// TIA Portal project "DALU-Projekt_HMI_V19" (V19)

(* hardware
DEVICE "SIMATIC 1200-Station_3"  S71200.Device
   slot 0: "S7-1200 Baugruppenträger"  Rack  V1.0
   slot 1: "Target_3"  CPU 1214C DC/DC/DC  6ES7 214-1AE30-0XB0  V2.2
   slot 101: "Target 3 CM 1243-2"  CM 1243-2  3RK7243-2AA30-0XB0  V1.0
   slot 102: "Target 3 CM 1243-5"  CM 1243-5  6GK7 243-5DX30-0XE0  V1.0
DEVICE "ASi-3-S9 (4DI)"  AS-i slave
   slot 0: "-"  Rail
   slot 1: "ASi-3-S9 (4DI)"  AS-i Standard Slave  AS-i Standard Slave Universal
      slot 1: "ASi-3-S9 (4DI) [AS-i Slave (D)]"  AS-i Address-Module
      slot 2: "ASi-3-S9 (4DI) [AS-i Slave (A)]"  AS-i Address-Module
      slot 3: "ASi-3-S9 (4DI) [AS-i Slave (T)]"  AS-i Address-Module
DEVICE "ASi-3-S5 (2AI)"  AS-i slave
   slot 0: "-"  Rail
   slot 1: "ASi-3-S5 (2AI)"  AS-i K60, 2AI-C  3RK1 207-1BQ40-0AA3
      slot 1: "ASi-3-S5 (2AI) [AS-i Slave (D)]"  AS-i Address-Module
      slot 2: "ASi-3-S5 (2AI) [AS-i Slave (A)]"  AS-i Address-Module
      slot 3: "ASi-3-S5 (2AI) [AS-i Slave (T)]"  AS-i Address-Module
DEVICE "ASi-3-S1 (4DI/4DO)"  AS-i slave
   slot 0: "-"  Rail
   slot 1: "ASi-3-S1 (4DI/4DO)"  AS-i 3SB3, 4DI/4DO  3SF5 500-0BC
      slot 1: "ASi-3-S1 (4DI/4DO) [AS-i Slave (D)]"  AS-i Address-Module
      slot 2: "ASi-3-S1 (4DI/4DO) [AS-i Slave (A)]"  AS-i Address-Module
      slot 3: "ASi-3-S1 (4DI/4DO) [AS-i Slave (T)]"  AS-i Address-Module
DEVICE "ASi-3-S7 (2DI,2PO)"  AS-i slave
   slot 0: "-"  Rail
   slot 1: "ASi-3-S7 (2DI,2PO)"  AS-i Standard Slave  AS-i Standard Slave Universal
      slot 1: "ASi-3-S7 (2DI,2PO) [AS-i Slave (D)]"  AS-i Address-Module
      slot 2: "ASi-3-S7 (2DI,2PO) [AS-i Slave (A)]"  AS-i Address-Module
      slot 3: "ASi-3-S7 (2DI,2PO) [AS-i Slave (T)]"  AS-i Address-Module
DEVICE "ASi-3-S3 (2AI)"  AS-i slave
   slot 0: "-"  Rail
   slot 1: "ASi-3-S3 (2AI)"  AS-i K60, 2AI-V  3RK1 207-2BQ40-0AA3
      slot 1: "ASi-3-S3 (2AI) [AS-i Slave (D)]"  AS-i Address-Module
      slot 2: "ASi-3-S3 (2AI) [AS-i Slave (A)]"  AS-i Address-Module
      slot 3: "ASi-3-S3 (2AI) [AS-i Slave (T)]"  AS-i Address-Module
DEVICE "ASi-3-S8 (3DI/1DO)"  AS-i slave
   slot 0: "-"  Rail
   slot 1: "ASi-3-S8 (3DI/1DO)"  AS-i Standard Slave  AS-i Standard Slave Universal
      slot 1: "ASi-3-S8 (3DI/1DO) [AS-i Slave (D)]"  AS-i Address-Module
      slot 2: "ASi-3-S8 (3DI/1DO) [AS-i Slave (A)]"  AS-i Address-Module
      slot 3: "ASi-3-S8 (3DI/1DO) [AS-i Slave (T)]"  AS-i Address-Module
DEVICE "DP_3_S1"  GSD.Device
   slot 0: "Baugruppenträger"  Rail
   slot 0: "DP_3_Simodrive"  6FX2001-5xPxx  4.2
DEVICE "ASi-3-S2 (2AO)"  AS-i slave
   slot 0: "-"  Rail
   slot 1: "ASi-3-S2 (2AO)"  AS-i K60, 2AO-V  3RK1 107-2BQ40-0AA3
      slot 1: "ASi-3-S2 (2AO) [AS-i Slave (D)]"  AS-i Address-Module
      slot 2: "ASi-3-S2 (2AO) [AS-i Slave (A)]"  AS-i Address-Module
      slot 3: "ASi-3-S2 (2AO) [AS-i Slave (T)]"  AS-i Address-Module
DEVICE "ASi-3-S4 (4DI/4DO)"  AS-i slave
   slot 0: "-"  Rail
   slot 1: "ASi-3-S4 (4DI/4DO)"  AS-i K60, 4DI/4DO  3RK1 400-1DQ01-0AA3
      slot 1: "ASi-3-S4 (4DI/4DO) [AS-i Slave (D)]"  AS-i Address-Module
      slot 2: "ASi-3-S4 (4DI/4DO) [AS-i Slave (A)]"  AS-i Address-Module
      slot 3: "ASi-3-S4 (4DI/4DO) [AS-i Slave (T)]"  AS-i Address-Module
DEVICE "ASi-3-S6 (4DI)"  AS-i slave
   slot 0: "-"  Rail
   slot 1: "ASi-3-S6 (4DI)"  AS-i K45, 4DI  3RK1 200-0CQ20-0AA3
      slot 1: "ASi-3-S6 (4DI) [AS-i Slave (D)]"  AS-i Address-Module
      slot 2: "ASi-3-S6 (4DI) [AS-i Slave (A)]"  AS-i Address-Module
      slot 3: "ASi-3-S6 (4DI) [AS-i Slave (T)]"  AS-i Address-Module
DEVICE "SIMATIC 1200-Station_4"  S71200.Device
   slot 0: "S7-1200 Baugruppenträger"  Rack  V1.0
   slot 1: "Target_4"  CPU 1214C DC/DC/DC  6ES7 214-1AE30-0XB0  V2.2
   slot 101: "Target 4 CM 1243-2"  CM 1243-2  3RK7243-2AA30-0XB0  V1.0
   slot 102: "Target 4 CM 1243-5"  CM 1243-5  6GK7 243-5DX30-0XE0  V1.0
DEVICE "ASi-4-S9 (4DI)"  AS-i slave
   slot 0: "-"  Rail
   slot 1: "ASi-4-S9 (4DI)"  AS-i Standard Slave  AS-i Standard Slave Universal
      slot 1: "ASi-4-S9 (4DI) [AS-i Slave (D)]"  AS-i Address-Module
      slot 2: "ASi-4-S9 (4DI) [AS-i Slave (A)]"  AS-i Address-Module
      slot 3: "ASi-4-S9 (4DI) [AS-i Slave (T)]"  AS-i Address-Module
DEVICE "ASi-4-S5 (2AI)"  AS-i slave
   slot 0: "-"  Rail
   slot 1: "ASi-4-S5 (2AI)"  AS-i K60, 2AI-C  3RK1 207-1BQ40-0AA3
      slot 1: "ASi-4-S5 (2AI) [AS-i Slave (D)]"  AS-i Address-Module
      slot 2: "ASi-4-S5 (2AI) [AS-i Slave (A)]"  AS-i Address-Module
      slot 3: "ASi-4-S5 (2AI) [AS-i Slave (T)]"  AS-i Address-Module
DEVICE "ASi-4-S1 (4DI/4DO)"  AS-i slave
   slot 0: "-"  Rail
   slot 1: "ASi-4-S1 (4DI/4DO)"  AS-i 3SB3, 4DI/4DO  3SF5 500-0BC
      slot 1: "ASi-4-S1 (4DI/4DO) [AS-i Slave (D)]"  AS-i Address-Module
      slot 2: "ASi-4-S1 (4DI/4DO) [AS-i Slave (A)]"  AS-i Address-Module
      slot 3: "ASi-4-S1 (4DI/4DO) [AS-i Slave (T)]"  AS-i Address-Module
DEVICE "ASi-4-S7 (2DI,2PO)"  AS-i slave
   slot 0: "-"  Rail
   slot 1: "ASi-4-S7 (2DI,2PO)"  AS-i Standard Slave  AS-i Standard Slave Universal
      slot 1: "ASi-4-S7 (2DI,2PO) [AS-i Slave (D)]"  AS-i Address-Module
      slot 2: "ASi-4-S7 (2DI,2PO) [AS-i Slave (A)]"  AS-i Address-Module
      slot 3: "ASi-4-S7 (2DI,2PO) [AS-i Slave (T)]"  AS-i Address-Module
DEVICE "ASi-4-S3 (2AI)"  AS-i slave
   slot 0: "-"  Rail
   slot 1: "ASi-4-S3 (2AI)"  AS-i K60, 2AI-V  3RK1 207-2BQ40-0AA3
      slot 1: "ASi-4-S3 (2AI) [AS-i Slave (D)]"  AS-i Address-Module
      slot 2: "ASi-4-S3 (2AI) [AS-i Slave (A)]"  AS-i Address-Module
      slot 3: "ASi-4-S3 (2AI) [AS-i Slave (T)]"  AS-i Address-Module
DEVICE "ASi-4-S8 (3DI/1DO)"  AS-i slave
   slot 0: "-"  Rail
   slot 1: "ASi-4-S8 (3DI/1DO)"  AS-i Standard Slave  AS-i Standard Slave Universal
      slot 1: "ASi-4-S8 (3DI/1DO) [AS-i Slave (D)]"  AS-i Address-Module
      slot 2: "ASi-4-S8 (3DI/1DO) [AS-i Slave (A)]"  AS-i Address-Module
      slot 3: "ASi-4-S8 (3DI/1DO) [AS-i Slave (T)]"  AS-i Address-Module
DEVICE "DP_4_S1"  GSD.Device
   slot 0: "Baugruppenträger"  Rail
   slot 0: "DP_4_Simodrive"  6FX2001-5xPxx  4.2
DEVICE "ASi-4-S2 (2AO)"  AS-i slave
   slot 0: "-"  Rail
   slot 1: "ASi-4-S2 (2AO)"  AS-i K60, 2AO-V  3RK1 107-2BQ40-0AA3
      slot 1: "ASi-4-S2 (2AO) [AS-i Slave (D)]"  AS-i Address-Module
      slot 2: "ASi-4-S2 (2AO) [AS-i Slave (A)]"  AS-i Address-Module
      slot 3: "ASi-4-S2 (2AO) [AS-i Slave (T)]"  AS-i Address-Module
DEVICE "ASi-4-S4 (4DI/4DO)"  AS-i slave
   slot 0: "-"  Rail
   slot 1: "ASi-4-S4 (4DI/4DO)"  AS-i K60, 4DI/4DO  3RK1 400-1DQ01-0AA3
      slot 1: "ASi-4-S4 (4DI/4DO) [AS-i Slave (D)]"  AS-i Address-Module
      slot 2: "ASi-4-S4 (4DI/4DO) [AS-i Slave (A)]"  AS-i Address-Module
      slot 3: "ASi-4-S4 (4DI/4DO) [AS-i Slave (T)]"  AS-i Address-Module
DEVICE "ASi-4-S6 (4DI)"  AS-i slave
   slot 0: "-"  Rail
   slot 1: "ASi-4-S6 (4DI)"  AS-i K45, 4DI  3RK1 200-0CQ20-0AA3
      slot 1: "ASi-4-S6 (4DI) [AS-i Slave (D)]"  AS-i Address-Module
      slot 2: "ASi-4-S6 (4DI) [AS-i Slave (A)]"  AS-i Address-Module
      slot 3: "ASi-4-S6 (4DI) [AS-i Slave (T)]"  AS-i Address-Module
DEVICE "SIMATIC 1200-Station_5"  S71200.Device
   slot 0: "S7-1200 Baugruppenträger"  Rack  V1.0
   slot 1: "Target_5"  CPU 1214C DC/DC/DC  6ES7 214-1AE30-0XB0  V2.2
   slot 101: "Target 5 CM 1243-2"  CM 1243-2  3RK7243-2AA30-0XB0  V1.0
   slot 102: "Target 5 CM 1243-5"  CM 1243-5  6GK7 243-5DX30-0XE0  V1.0
   slot 103: "CM CANopen_1"  021620-B  V1.0
DEVICE "ASi-5-S9 (4DI)"  AS-i slave
   slot 0: "-"  Rail
   slot 1: "ASi-5-S9 (4DI)"  AS-i Standard Slave  AS-i Standard Slave Universal
      slot 1: "ASi-5-S9 (4DI) [AS-i Slave (D)]"  AS-i Address-Module
      slot 2: "ASi-5-S9 (4DI) [AS-i Slave (A)]"  AS-i Address-Module
      slot 3: "ASi-5-S9 (4DI) [AS-i Slave (T)]"  AS-i Address-Module
DEVICE "ASi-5-S5 (2AI)"  AS-i slave
   slot 0: "-"  Rail
   slot 1: "ASi-5-S5 (2AI)"  AS-i K60, 2AI-C  3RK1 207-1BQ40-0AA3
      slot 1: "ASi-5-S5 (2AI) [AS-i Slave (D)]"  AS-i Address-Module
      slot 2: "ASi-5-S5 (2AI) [AS-i Slave (A)]"  AS-i Address-Module
      slot 3: "ASi-5-S5 (2AI) [AS-i Slave (T)]"  AS-i Address-Module
DEVICE "ASi-5-S3 (2AI)"  AS-i slave
   slot 0: "-"  Rail
   slot 1: "ASi-5-S3 (2AI)"  AS-i K60, 2AI-V  3RK1 207-2BQ40-0AA3
      slot 1: "ASi-5-S3 (2AI) [AS-i Slave (D)]"  AS-i Address-Module
      slot 2: "ASi-5-S3 (2AI) [AS-i Slave (A)]"  AS-i Address-Module
      slot 3: "ASi-5-S3 (2AI) [AS-i Slave (T)]"  AS-i Address-Module
DEVICE "ASi-5-S7 (2DI,2PO)"  AS-i slave
   slot 0: "-"  Rail
   slot 1: "ASi-5-S7 (2DI,2PO)"  AS-i Standard Slave  AS-i Standard Slave Universal
      slot 1: "ASi-5-S7 (2DI,2PO) [AS-i Slave (D)]"  AS-i Address-Module
      slot 2: "ASi-5-S7 (2DI,2PO) [AS-i Slave (A)]"  AS-i Address-Module
      slot 3: "ASi-5-S7 (2DI,2PO) [AS-i Slave (T)]"  AS-i Address-Module
DEVICE "ASi-5-S2 (2AO)"  AS-i slave
   slot 0: "-"  Rail
   slot 1: "ASi-5-S2 (2AO)"  AS-i K60, 2AO-V  3RK1 107-2BQ40-0AA3
      slot 1: "ASi-5-S2 (2AO) [AS-i Slave (D)]"  AS-i Address-Module
      slot 2: "ASi-5-S2 (2AO) [AS-i Slave (A)]"  AS-i Address-Module
      slot 3: "ASi-5-S2 (2AO) [AS-i Slave (T)]"  AS-i Address-Module
DEVICE "ASi-5-S8 (3DI/1DO)"  AS-i slave
   slot 0: "-"  Rail
   slot 1: "ASi-5-S8 (3DI/1DO)"  AS-i Standard Slave  AS-i Standard Slave Universal
      slot 1: "ASi-5-S8 (3DI/1DO) [AS-i Slave (D)]"  AS-i Address-Module
      slot 2: "ASi-5-S8 (3DI/1DO) [AS-i Slave (A)]"  AS-i Address-Module
      slot 3: "ASi-5-S8 (3DI/1DO) [AS-i Slave (T)]"  AS-i Address-Module
DEVICE "ASi-5-S1 (4DI/4DO)"  AS-i slave
   slot 0: "-"  Rail
   slot 1: "ASi-5-S1 (4DI/4DO)"  AS-i 3SB3, 4DI/4DO  3SF5 500-0BC
      slot 1: "ASi-5-S1 (4DI/4DO) [AS-i Slave (D)]"  AS-i Address-Module
      slot 2: "ASi-5-S1 (4DI/4DO) [AS-i Slave (A)]"  AS-i Address-Module
      slot 3: "ASi-5-S1 (4DI/4DO) [AS-i Slave (T)]"  AS-i Address-Module
DEVICE "DP_5_S1"  GSD.Device
   slot 0: "Baugruppenträger"  Rail
   slot 0: "DP_5_Simodrive"  6FX2001-5xPxx  4.2
DEVICE "ASi-5-S4 (4DI/4DO)"  AS-i slave
   slot 0: "-"  Rail
   slot 1: "ASi-5-S4 (4DI/4DO)"  AS-i K60, 4DI/4DO  3RK1 400-1DQ01-0AA3
      slot 1: "ASi-5-S4 (4DI/4DO) [AS-i Slave (D)]"  AS-i Address-Module
      slot 2: "ASi-5-S4 (4DI/4DO) [AS-i Slave (A)]"  AS-i Address-Module
      slot 3: "ASi-5-S4 (4DI/4DO) [AS-i Slave (T)]"  AS-i Address-Module
DEVICE "ASi-5-S6 (4DI)"  AS-i slave
   slot 0: "-"  Rail
   slot 1: "ASi-5-S6 (4DI)"  AS-i K45, 4DI  3RK1 200-0CQ20-0AA3
      slot 1: "ASi-5-S6 (4DI) [AS-i Slave (D)]"  AS-i Address-Module
      slot 2: "ASi-5-S6 (4DI) [AS-i Slave (A)]"  AS-i Address-Module
      slot 3: "ASi-5-S6 (4DI) [AS-i Slave (T)]"  AS-i Address-Module
DEVICE "SIMATIC 1200-Station_1"  S71200.Device
   slot 0: "S7-1200 Baugruppenträger"  Rack  V1.0
   slot 1: "Target_1"  CPU 1214C DC/DC/DC  6ES7 214-1AE30-0XB0  V2.2
   slot 101: "Target 1 CM 1243-2"  CM 1243-2  3RK7243-2AA30-0XB0  V1.0
   slot 102: "Target 1 CM 1243-5"  CM 1243-5  6GK7 243-5DX30-0XE0  V1.0
DEVICE "ASi-1-S1 (4DI/4DO)"  AS-i slave
   slot 0: "-"  Rail
   slot 1: "ASi-1-S1 (4DI/4DO)"  AS-i 3SB3, 4DI/4DO  3SF5 500-0BC
      slot 1: "ASi-1-S1 (4DI/4DO) [AS-i Slave (D)]"  AS-i Address-Module
      slot 2: "ASi-1-S1 (4DI/4DO) [AS-i Slave (A)]"  AS-i Address-Module
      slot 3: "ASi-1-S1 (4DI/4DO) [AS-i Slave (T)]"  AS-i Address-Module
DEVICE "DP_1_S1"  GSD.Device
   slot 0: "Baugruppenträger"  Rail
   slot 0: "DP_1_Simodrive"  6FX2001-5xPxx  4.2
DEVICE "ASi-1-S4 (4DI/4DO)"  AS-i slave
   slot 0: "-"  Rail
   slot 1: "ASi-1-S4 (4DI/4DO)"  AS-i K60, 4DI/4DO  3RK1 400-1DQ01-0AA3
      slot 1: "ASi-1-S4 (4DI/4DO) [AS-i Slave (D)]"  AS-i Address-Module
      slot 2: "ASi-1-S4 (4DI/4DO) [AS-i Slave (A)]"  AS-i Address-Module
      slot 3: "ASi-1-S4 (4DI/4DO) [AS-i Slave (T)]"  AS-i Address-Module
DEVICE "ASi-1-S6 (4DI)"  AS-i slave
   slot 0: "-"  Rail
   slot 1: "ASi-1-S6 (4DI)"  AS-i K45, 4DI  3RK1 200-0CQ20-0AA3
      slot 1: "ASi-1-S6 (4DI) [AS-i Slave (D)]"  AS-i Address-Module
      slot 2: "ASi-1-S6 (4DI) [AS-i Slave (A)]"  AS-i Address-Module
      slot 3: "ASi-1-S6 (4DI) [AS-i Slave (T)]"  AS-i Address-Module
DEVICE "ASi-1-S9 (4DI)"  AS-i slave
   slot 0: "-"  Rail
   slot 1: "ASi-1-S9 (4DI)"  AS-i Standard Slave  AS-i Standard Slave Universal
      slot 1: "ASi-1-S9 (4DI) [AS-i Slave (D)]"  AS-i Address-Module
      slot 2: "ASi-1-S9 (4DI) [AS-i Slave (A)]"  AS-i Address-Module
      slot 3: "ASi-1-S9 (4DI) [AS-i Slave (T)]"  AS-i Address-Module
DEVICE "ASi-1-S5 (2AI)"  AS-i slave
   slot 0: "-"  Rail
   slot 1: "ASi-1-S5 (2AI)"  AS-i K60, 2AI-C  3RK1 207-1BQ40-0AA3
      slot 1: "ASi-1-S5 (2AI) [AS-i Slave (D)]"  AS-i Address-Module
      slot 2: "ASi-1-S5 (2AI) [AS-i Slave (A)]"  AS-i Address-Module
      slot 3: "ASi-1-S5 (2AI) [AS-i Slave (T)]"  AS-i Address-Module
DEVICE "ASi-1-S3 (2AI)"  AS-i slave
   slot 0: "-"  Rail
   slot 1: "ASi-1-S3 (2AI)"  AS-i K60, 2AI-V  3RK1 207-2BQ40-0AA3
      slot 1: "ASi-1-S3 (2AI) [AS-i Slave (D)]"  AS-i Address-Module
      slot 2: "ASi-1-S3 (2AI) [AS-i Slave (A)]"  AS-i Address-Module
      slot 3: "ASi-1-S3 (2AI) [AS-i Slave (T)]"  AS-i Address-Module
DEVICE "ASi-1-S7 (2DI,2PO)"  AS-i slave
   slot 0: "-"  Rail
   slot 1: "ASi-1-S7 (2DI,2PO)"  AS-i Standard Slave  AS-i Standard Slave Universal
      slot 1: "ASi-1-S7 (2DI,2PO) [AS-i Slave (D)]"  AS-i Address-Module
      slot 2: "ASi-1-S7 (2DI,2PO) [AS-i Slave (A)]"  AS-i Address-Module
      slot 3: "ASi-1-S7 (2DI,2PO) [AS-i Slave (T)]"  AS-i Address-Module
DEVICE "ASi-1-S2 (2AO)"  AS-i slave
   slot 0: "-"  Rail
   slot 1: "ASi-1-S2 (2AO)"  AS-i K60, 2AO-V  3RK1 107-2BQ40-0AA3
      slot 1: "ASi-1-S2 (2AO) [AS-i Slave (D)]"  AS-i Address-Module
      slot 2: "ASi-1-S2 (2AO) [AS-i Slave (A)]"  AS-i Address-Module
      slot 3: "ASi-1-S2 (2AO) [AS-i Slave (T)]"  AS-i Address-Module
DEVICE "ASi-1-S8 (3DI/1DO)"  AS-i slave
   slot 0: "-"  Rail
   slot 1: "ASi-1-S8 (3DI/1DO)"  AS-i Standard Slave  AS-i Standard Slave Universal
      slot 1: "ASi-1-S8 (3DI/1DO) [AS-i Slave (D)]"  AS-i Address-Module
      slot 2: "ASi-1-S8 (3DI/1DO) [AS-i Slave (A)]"  AS-i Address-Module
      slot 3: "ASi-1-S8 (3DI/1DO) [AS-i Slave (T)]"  AS-i Address-Module
DEVICE "ASi-2-S8 (3DI/1DO)"  AS-i slave
   slot 0: "-"  Rail
   slot 1: "ASi-2-S8 (3DI/1DO)"  AS-i Standard Slave  AS-i Standard Slave Universal
      slot 1: "ASi-2-S8 (3DI/1DO) [AS-i Slave (D)]"  AS-i Address-Module
      slot 2: "ASi-2-S8 (3DI/1DO) [AS-i Slave (A)]"  AS-i Address-Module
      slot 3: "ASi-2-S8 (3DI/1DO) [AS-i Slave (T)]"  AS-i Address-Module
DEVICE "ASi-2-S2 (2AO)"  AS-i slave
   slot 0: "-"  Rail
   slot 1: "ASi-2-S2 (2AO)"  AS-i K60, 2AO-V  3RK1 107-2BQ40-0AA3
      slot 1: "ASi-2-S2 (2AO) [AS-i Slave (D)]"  AS-i Address-Module
      slot 2: "ASi-2-S2 (2AO) [AS-i Slave (A)]"  AS-i Address-Module
      slot 3: "ASi-2-S2 (2AO) [AS-i Slave (T)]"  AS-i Address-Module
DEVICE "ASi-2-S7 (2DI,2PO)"  AS-i slave
   slot 0: "-"  Rail
   slot 1: "ASi-2-S7 (2DI,2PO)"  AS-i Standard Slave  AS-i Standard Slave Universal
      slot 1: "ASi-2-S7 (2DI,2PO) [AS-i Slave (D)]"  AS-i Address-Module
      slot 2: "ASi-2-S7 (2DI,2PO) [AS-i Slave (A)]"  AS-i Address-Module
      slot 3: "ASi-2-S7 (2DI,2PO) [AS-i Slave (T)]"  AS-i Address-Module
DEVICE "ASi-2-S3 (2AI)"  AS-i slave
   slot 0: "-"  Rail
   slot 1: "ASi-2-S3 (2AI)"  AS-i K60, 2AI-V  3RK1 207-2BQ40-0AA3
      slot 1: "ASi-2-S3 (2AI) [AS-i Slave (D)]"  AS-i Address-Module
      slot 2: "ASi-2-S3 (2AI) [AS-i Slave (A)]"  AS-i Address-Module
      slot 3: "ASi-2-S3 (2AI) [AS-i Slave (T)]"  AS-i Address-Module
DEVICE "ASi-2-S5 (2AI)"  AS-i slave
   slot 0: "-"  Rail
   slot 1: "ASi-2-S5 (2AI)"  AS-i K60, 2AI-C  3RK1 207-1BQ40-0AA3
      slot 1: "ASi-2-S5 (2AI) [AS-i Slave (D)]"  AS-i Address-Module
      slot 2: "ASi-2-S5 (2AI) [AS-i Slave (A)]"  AS-i Address-Module
      slot 3: "ASi-2-S5 (2AI) [AS-i Slave (T)]"  AS-i Address-Module
DEVICE "ASi-2-S9 (4DI)"  AS-i slave
   slot 0: "-"  Rail
   slot 1: "ASi-2-S9 (4DI)"  AS-i Standard Slave  AS-i Standard Slave Universal
      slot 1: "ASi-2-S9 (4DI) [AS-i Slave (D)]"  AS-i Address-Module
      slot 2: "ASi-2-S9 (4DI) [AS-i Slave (A)]"  AS-i Address-Module
      slot 3: "ASi-2-S9 (4DI) [AS-i Slave (T)]"  AS-i Address-Module
DEVICE "ASi-2-S4 (4DI/4DO)"  AS-i slave
   slot 0: "-"  Rail
   slot 1: "ASi-2-S4 (4DI/4DO)"  AS-i K60, 4DI/4DO  3RK1 400-1DQ01-0AA3
      slot 1: "ASi-2-S4 (4DI/4DO) [AS-i Slave (D)]"  AS-i Address-Module
      slot 2: "ASi-2-S4 (4DI/4DO) [AS-i Slave (A)]"  AS-i Address-Module
      slot 3: "ASi-2-S4 (4DI/4DO) [AS-i Slave (T)]"  AS-i Address-Module
DEVICE "DP_2_S1"  GSD.Device
   slot 0: "Baugruppenträger"  Rail
   slot 0: "DP_2_Simodrive"  6FX2001-5xPxx  4.2
DEVICE "ASi-2-S1 (4DI/4DO)"  AS-i slave
   slot 0: "-"  Rail
   slot 1: "ASi-2-S1 (4DI/4DO)"  AS-i 3SB3, 4DI/4DO  3SF5 500-0BC
      slot 1: "ASi-2-S1 (4DI/4DO) [AS-i Slave (D)]"  AS-i Address-Module
      slot 2: "ASi-2-S1 (4DI/4DO) [AS-i Slave (A)]"  AS-i Address-Module
      slot 3: "ASi-2-S1 (4DI/4DO) [AS-i Slave (T)]"  AS-i Address-Module
DEVICE "SIMATIC 1200-Station_2"  S71200.Device
   slot 0: "S7-1200 Baugruppenträger"  Rack  V1.0
   slot 1: "Target_2"  CPU 1214C DC/DC/DC  6ES7 214-1AE30-0XB0  V2.2
   slot 101: "Target 2 CM 1243-2"  CM 1243-2  3RK7243-2AA30-0XB0  V1.0
   slot 102: "Target 2 CM 1243-5"  CM 1243-5  6GK7 243-5DX30-0XE0  V1.0
DEVICE "ASi-2-S6 (4DI)"  AS-i slave
   slot 0: "-"  Rail
   slot 1: "ASi-2-S6 (4DI)"  AS-i K45, 4DI, A/B  3RK2 200-0CQ20-0AA3
      slot 1: "ASi-2-S6 (4DI) [AS-i Slave (D)]"  AS-i Address-Module
      slot 2: "ASi-2-S6 (4DI) [AS-i Slave (A)]"  AS-i Address-Module
      slot 3: "ASi-2-S6 (4DI) [AS-i Slave (T)]"  AS-i Address-Module
DEVICE "HMI_1"  KTP400 Comfort
   slot 0: "HMI_1"  KTP400 Comfort  6AV2 124-2DC01-0AX0  15.1.0.0
   slot 1: "HMI_RT_1"  KTP400 Comfort  6AV2 124-2DC01-0AX0  15.1.0.0
   slot 5: "HMI_1.IE_CP_1"  PROFINET Interface  15.0.1.0
      slot 1: "PROFINET Interface_1"  PROFINET Interface
         slot 1: "Port_1"  Port
   slot 7: "HMI_1.MPI/DP_CP_1"  MPI/DP Interface  15.0.1.0
DEVICE "HMI_2"  KTP400 Comfort
   slot 0: "HMI_1"  KTP400 Comfort  6AV2 124-2DC01-0AX0  15.1.0.0
   slot 1: "HMI_RT_2"  KTP400 Comfort  6AV2 124-2DC01-0AX0  15.1.0.0
   slot 5: "HMI_1.IE_CP_1"  PROFINET Interface  15.0.1.0
      slot 1: "PROFINET Interface_1"  PROFINET Interface
         slot 1: "Port_1"  Port
   slot 7: "HMI_1.MPI/DP_CP_1"  MPI/DP Interface  15.0.1.0
DEVICE "HMI_3"  KTP400 Comfort
   slot 0: "HMI_1"  KTP400 Comfort  6AV2 124-2DC01-0AX0  15.1.0.0
   slot 1: "HMI_RT_3"  KTP400 Comfort  6AV2 124-2DC01-0AX0  15.1.0.0
   slot 5: "HMI_1.IE_CP_1"  PROFINET Interface  15.0.1.0
      slot 1: "PROFINET Interface_1"  PROFINET Interface
         slot 1: "Port_1"  Port
   slot 7: "HMI_1.MPI/DP_CP_1"  MPI/DP Interface  15.0.1.0
DEVICE "HMI_4"  KTP400 Comfort
   slot 0: "HMI_1"  KTP400 Comfort  6AV2 124-2DC01-0AX0  15.1.0.0
   slot 1: "HMI_RT_4"  KTP400 Comfort  6AV2 124-2DC01-0AX0  15.1.0.0
   slot 5: "HMI_1.IE_CP_1"  PROFINET Interface  15.0.1.0
      slot 1: "PROFINET Interface_1"  PROFINET Interface
         slot 1: "Port_1"  Port
   slot 7: "HMI_1.MPI/DP_CP_1"  MPI/DP Interface  15.0.1.0
DEVICE "HMI_5"  KTP400 Comfort
   slot 0: "HMI_1"  KTP400 Comfort  6AV2 124-2DC01-0AX0  15.1.0.0
   slot 1: "HMI_RT_5"  KTP400 Comfort  6AV2 124-2DC01-0AX0  15.1.0.0
   slot 5: "HMI_1.IE_CP_1"  PROFINET Interface  15.0.1.0
      slot 1: "PROFINET Interface_1"  PROFINET Interface
         slot 1: "Port_1"  Port
   slot 7: "HMI_1.MPI/DP_CP_1"  MPI/DP Interface  15.0.1.0
*)

// ===== PLC "Target_3"  CPU 1214C DC/DC/DC =====

VAR_GLOBAL   // PLC tag table "Standard-Variablentabelle"
   "Swt0" AT %I0.0 : Bool;
   "Swt1" AT %I0.1 : Bool;
   "Swt2" AT %I0.2 : Bool;
   "Swt3" AT %I0.3 : Bool;
   "Swt4" AT %I0.4 : Bool;
   "Swt5" AT %I0.5 : Bool;
   "Swt6" AT %I0.6 : Bool;
   "Swt7" AT %I0.7 : Bool;
   "Swt0-7" AT %IB0 : Byte;
   "JOY_LeftRight" AT %IW70 : Int;
   "JOY_UpDown" AT %IW68 : Int;
   "MagE_D" AT %I7.1 : Bool;
   "MagE_U" AT %I7.2 : Bool;
   "Tast_1" AT %I2.2 : Bool;
   "LED0" AT %Q0.0 : Bool;
   "LED1" AT %Q0.1 : Bool;
   "LED2" AT %Q0.2 : Bool;
   "LED3" AT %Q0.3 : Bool;
   "LED4" AT %Q0.4 : Bool;
   "LED5" AT %Q0.5 : Bool;
   "LED6" AT %Q0.6 : Bool;
   "LED7" AT %Q0.7 : Bool;
   "LED0-7" AT %QB0 : Byte;
   "Lampe_0" AT %Q2.0 : Bool;
   "MCGO" AT %Q5.2 : Bool;
   "MCDIR" AT %Q5.3 : Bool;
   "MCSPEED" AT %QW66 : Word;
   "Lampe_1" AT %Q2.1 : Bool;
   "Lampe_2" AT %Q2.2 : Bool;
   "Clock_2.5Hz" AT %M8000.2 : Bool;
   "Clock_2Hz" AT %M8000.3 : Bool;
   "Clock_1.25Hz" AT %M8000.4 : Bool;
   "Clock_1Hz" AT %M8000.5 : Bool;
   "Clock_0.625Hz" AT %M8000.6 : Bool;
   "Clock_0.5Hz" AT %M8000.7 : Bool;
   "System_Byte" AT %MB8001 : Byte;
   "FirstScan" AT %M8001.0 : Bool;
   "AlwaysTRUE" AT %M8001.2 : Bool;
   "AlwaysFALSE" AT %M8001.3 : Bool;
   "IndNS_R" AT %M8002.0 : Bool;
END_VAR

DATA_BLOCK "DB_State"   // DB1
{ S7_Optimized_Access := 'TRUE' }
VERSION : 0.1
   VAR
      State : Int;
   END_VAR
BEGIN
END_DATA_BLOCK

DATA_BLOCK "DB_Materialerkennung"   // DB3
{ S7_Optimized_Access := 'TRUE' }
VERSION : 0.1
BEGIN
END_DATA_BLOCK

// folder: System blocks/Program resources

DATA_BLOCK "Timer_3.2"   // DB2
{ S7_Optimized_Access := 'TRUE' }
AUTHOR : Simatic
FAMILY : IEC
NAME : IEC_TMR
VERSION : 1.0
// stored: InstanceOfName IEC_TIMER
"IEC_TIMER"
BEGIN
END_DATA_BLOCK

// folder: (top level)

FUNCTION "Bsp3.1" : Void   // FC1, SCL
{ S7_Optimized_Access := 'TRUE' }
VERSION : 0.1
BEGIN
   IF "Swt0-7" <= 27 THEN
       "LED0-7" := "Swt0-7";
       ;
   ELSE
       "LED0-7" := 0;
   END_IF;
END_FUNCTION

FUNCTION "Bsp3.2" : Void   // FC2, SCL
{ S7_Optimized_Access := 'TRUE' }
VERSION : 0.1
BEGIN

   "Lampe_0" := "Clock_1Hz";
END_FUNCTION

FUNCTION "Bsp3.2_mit_timer" : Void   // FC3, SCL
{ S7_Optimized_Access := 'TRUE' }
VERSION : 0.1
BEGIN
   "Timer_3.2".TP(IN:="Clock_1Hz",
                  PT:=T#250ms,
                  Q=>"Lampe_0");
END_FUNCTION

FUNCTION "Bsp3.3" : Void   // FC4, SCL
{ S7_Optimized_Access := 'TRUE' }
VERSION : 0.1
   VAR CONSTANT
      JOY_MAX : Int := 1500;
      JOY_MIN : Int := -1500;
      JOY_MITTE : Int := 50;
   END_VAR
BEGIN
   IF "JOY_LeftRight" < 0.9 * #JOY_MIN THEN
       "LED3" := FALSE;
       "LED4" := FALSE;
       "LED5" := FALSE;
       "LED6" := TRUE;
   ELSIF "JOY_LeftRight" < 0.6 * #JOY_MIN THEN
       "LED3" := FALSE;
       "LED4" := FALSE;
       "LED5" := TRUE;
       "LED6" := FALSE;
   ELSIF "JOY_LeftRight" < 0.3 * #JOY_MIN THEN
       "LED3" := FALSE;
       "LED4" := TRUE;
       "LED5" := FALSE;
       "LED6" := FALSE;
   ELSIF "JOY_LeftRight" >= 0.3 * #JOY_MIN AND "JOY_LeftRight" <= #JOY_MITTE THEN
       "LED3" := TRUE;
       "LED4" := FALSE;
       "LED5" := FALSE;
       "LED6" := FALSE;
   ELSE
       "LED3" := FALSE;
       "LED4" := FALSE;
       "LED5" := FALSE;
       "LED6" := FALSE;
   END_IF;
END_FUNCTION

FUNCTION "Bsp3.4" : Void   // FC5, SCL
{ S7_Optimized_Access := 'TRUE' }
VERSION : 0.1
   VAR CONSTANT
      INT_MAX : Int := 16#FFFF;
   END_VAR
BEGIN
   //"MCSPEED" := #INT_MAX

   IF "DB_State".State = 0 THEN
       IF "MagE_D" = TRUE THEN
           "MCDIR" := 0;
           "DB_State".State := 1;
       ELSE
           "MCDIR" := 1;
           "DB_State".State := 2;
       END_IF;

   ELSIF "DB_State".State = 1 THEN
       "MCDIR" := 0;
       IF "MagE_U" = TRUE THEN
           "MCDIR" := 1;
           "DB_State".State := 2;

       END_IF;

   ELSIF "DB_State".State = 2 THEN
       "MCDIR" := 1;
       IF "MagE_D" = TRUE THEN
           "MCDIR" := 0;
           "DB_State".State := 1;

       END_IF;
   END_IF;

   IF "Swt7" THEN
       "MCGO" := TRUE;
       "Lampe_1" := FALSE;
       "Lampe_2" := TRUE;
      /// "DB_State".State := 0;
   ELSE
       "Lampe_1" := TRUE;
       "Lampe_2" := FALSE;
       "MCGO" := FALSE;
       //"DB_State".State := 10;
   END_IF;
END_FUNCTION

FUNCTION "Materialerkennung" : Void   // FC6, SCL
{ S7_Optimized_Access := 'TRUE' }
VERSION : 0.1
BEGIN
END_FUNCTION

ORGANIZATION_BLOCK "Main"   // OB1, SCL, ProgramCycle
TITLE = "Main Program Sweep (Cycle)"
{ S7_Optimized_Access := 'TRUE' }
VERSION : 0.1
BEGIN
   "Bsp3.1"();
   "Bsp3.2_mit_timer"();
   "Bsp3.3"();
   "Bsp3.4"();
END_ORGANIZATION_BLOCK

// ===== PLC "Target_4"  CPU 1214C DC/DC/DC =====

VAR_GLOBAL   // PLC tag table "Standard-Variablentabelle"
   "Clock_2.5Hz" AT %M8000.2 : Bool;
   "Clock_2Hz" AT %M8000.3 : Bool;
   "Clock_1.25Hz" AT %M8000.4 : Bool;
   "Clock_1Hz" AT %M8000.5 : Bool;
   "Clock_0.625Hz" AT %M8000.6 : Bool;
   "Clock_0.5Hz" AT %M8000.7 : Bool;
   "System_Byte" AT %MB8001 : Byte;
   "FirstScan" AT %M8001.0 : Bool;
   "AlwaysTRUE" AT %M8001.2 : Bool;
   "AlwaysFALSE" AT %M8001.3 : Bool;
END_VAR

ORGANIZATION_BLOCK "Main"   // OB1, LAD, ProgramCycle
TITLE = "Main Program Sweep (Cycle)"
{ S7_Optimized_Access := 'TRUE' }
VERSION : 0.1
BEGIN
END_ORGANIZATION_BLOCK

// ===== PLC "Target_5"  CPU 1214C DC/DC/DC =====

VAR_GLOBAL   // PLC tag table "Standard-Variablentabelle"
   "Swt0" AT %I0.0 : Bool;
   "Swt1" AT %I0.1 : Bool;
   "Swt2" AT %I0.2 : Bool;
   "Swt3" AT %I0.3 : Bool;
   "Swt4" AT %I0.4 : Bool;
   "Swt5" AT %I0.5 : Bool;
   "Swt6" AT %I0.6 : Bool;
   "Swt7" AT %I0.7 : Bool;
   "Swt0-7" AT %IB0 : Byte;
   "JOY_LeftRight" AT %IW70 : Int;
   "JOY_UpDown" AT %IW68 : Int;
   "MagE_D" AT %I7.1 : Bool;
   "MagE_U" AT %I7.2 : Bool;
   "LED0" AT %Q0.0 : Bool;
   "LED1" AT %Q0.1 : Bool;
   "LED2" AT %Q0.2 : Bool;
   "LED3" AT %Q0.3 : Bool;
   "LED4" AT %Q0.4 : Bool;
   "LED5" AT %Q0.5 : Bool;
   "LED6" AT %Q0.6 : Bool;
   "LED7" AT %Q0.7 : Bool;
   "LED0-7" AT %QB0 : Byte;
   "Lampe_0" AT %Q2.0 : Bool;
   "MCGO" AT %Q5.2 : Bool;
   "MCDIR" AT %Q5.3 : Bool;
   "MCSPEED" AT %QW66 : Word;
   "Lampe_1" AT %Q2.1 : Bool;
   "Lampe_2" AT %Q2.2 : Bool;
   "Clock_2.5Hz" AT %M8000.2 : Bool;
   "Clock_2Hz" AT %M8000.3 : Bool;
   "Clock_1.25Hz" AT %M8000.4 : Bool;
   "Clock_1Hz" AT %M8000.5 : Bool;
   "Clock_0.625Hz" AT %M8000.6 : Bool;
   "Clock_0.5Hz" AT %M8000.7 : Bool;
   "System_Byte" AT %MB8001 : Byte;
   "FirstScan" AT %M8001.0 : Bool;
   "AlwaysTRUE" AT %M8001.2 : Bool;
   "AlwaysFALSE" AT %M8001.3 : Bool;
   "IndNS_SS" AT %E9.0 : Bool;
   "IndNS_SSV" AT %E9.1 : Bool;
   "IndNS_OS" AT %I9.2 : Bool;
   "Dist" AT %EW74 : Word;
   "Druck" AT %EW72 : Word;
   "KapNS" AT %E5.2 : Bool;
   "ElMag" AT %A1.1 : Bool;
   "OptNS" AT %E5.3 : Bool;
   "ZendUP" AT %E8.1 : Bool;
   "ZendDO" AT %E8.0 : Bool;
   "Button_0" AT %E2.0 : Bool;
   "Button_1" AT %I2.1 : Bool;
   "Button_2" AT %E2.2 : Bool;
   "Button_3" AT %E2.3 : Bool;
   "ZylUp" AT %Q8.3 : Bool;
   "ZylDown" AT %Q8.2 : Bool;
   "Lampe_3" AT %A2.3 : Bool;
   "GlasLS" AT %E7.0 : Bool;
   "EinLS" AT %I5.0 : Bool;
   "Sonar_1" AT %E10.0 : Bool;
   "Sonar_2" AT %E10.1 : Bool;
   "Sonar_3" AT %E10.2 : Bool;
END_VAR

VAR_GLOBAL CONSTANT   // PLC tag table "Standard-Variablentabelle"
   "INIT" : UInt := 0;
   "START" : UInt := 2;
   "OCCUPIED" : UInt := 6;
   "TEST" : UInt := 7;
   "RESET" : UInt := 9;
   "COATING_A" : UInt := 10;
   "COATING_B" : UInt := 11;
   "COATING_C" : UInt := 12;
   "tank1_dist" : Int := 22400;
   "tank2_dist" : Int := 14200;
   "tank3_dist" : Int := 11200;
   "tank4_dist" : Int := 8550;
   "MANUAL" : UInt := 1;
   "Joy_Up" : Int := 1000;
   "Joy_Down" : Int := -1000;
   "ERROR" : UInt := 3;
END_VAR

// folder: CANOpen

TYPE "PIInput_CANOpen"
VERSION : 0.1
   STRUCT
      PIIn : Struct
         TempLo : Byte;
         TempHi : Byte;
      END_STRUCT;
   END_STRUCT;
END_TYPE

TYPE "SDO_ReadData"
VERSION : 0.1
   STRUCT
      SDO_ReadData : Array[1..245] of Byte;
   END_STRUCT;
END_TYPE

TYPE "SDO_WriteData"
VERSION : 0.1
   STRUCT
      SDO_WriteData : Array[1..245] of Byte;
   END_STRUCT;
END_TYPE

// folder: (top level)

DATA_BLOCK "DB_State"   // DB1
{ S7_Optimized_Access := 'TRUE' }
VERSION : 0.1
   VAR
      TimerFlag : Bool;
      "Timer" : Time;
      State : UInt;
   END_VAR
BEGIN
END_DATA_BLOCK

DATA_BLOCK "Block_1_DB"   // DB4
{ S7_Optimized_Access := 'TRUE' }
VERSION : 0.1
// stored: InstanceOfName Block_1
"Block_1"
BEGIN
END_DATA_BLOCK

DATA_BLOCK "CANopenProcessImage"   // DB14
TITLE = process image data of the CM in the format expected by the PLC
{ S7_Optimized_Access := 'FALSE' }
VERSION : 0.1
// DB provides the process image input / output data of the CM module but in the format of the PLC so the PLC can access them with the variable name.
   VAR
      ByteSize_PIInput_CANopen : UInt;   // byte size of the structure "PIInput_CANopen"
      CM_PIInput : "PIInput_CANOpen";   // uploaded pi input is copied to this structure
      PLC_PIInput : "PIInput_CANOpen";   // updated and converted pi input for the application
   END_VAR
BEGIN
END_DATA_BLOCK

// folder: CM CANopen

DATA_BLOCK "Ctrl_CM_CANopen"   // DB7
{ S7_Optimized_Access := 'FALSE' }
VERSION : 0.1
   VAR
      HW_ID : Hw_Io;   // hardware identifier of the accessed CM module
      GetNNStatus : Struct   // management of "Get Node & Network Status"
         fREQ : Bool := FALSE;   // TRUE: run "Get Node & Network Status" command
         abData : Array[0..131] of Byte;   // data array that this updated by "Get Node & Network Status"
      END_STRUCT;
      GetPIIn : Struct   // management of "Get Process Data In"
         fReq : Bool := FALSE;
      END_STRUCT;
      SetPIOut : Struct   // management of "Set Process Data Out"
         fReq : Bool := FALSE;   // TRUE: run SetProcessDataOut [FC3]
         fUpdateData : Bool := TRUE;   // "state machine" of SetProcessDataOut [FC3]: default: TRUE
      END_STRUCT;
      WriteSDO : Struct   // management of a SDO write command
         fREQ : Bool := FALSE;   // flag controls REQ input of WriteSDO FB
         HW_ID : Hw_Io;   // hardware identifier of the accessed CM module in TIA Portal
         bSLOT : Byte;   // selected SLOT number
         iNODE : Int;   // CANopen node id of the accessed device
         wINDEX : Word;   // accessed index of the object dictionary
         bSUB : Byte;   // accessed subindex of the object dictionary
         uiSIZE : UInt;   // number of data bytes to be written
         fBusy : Bool;   // variable keeps the value of output BUSY of WriteSDO FB
         uiRet : UInt;   // variable keeps the value of output RET of WriteSDO FB
         Data : "SDO_WriteData";   // data area where to get the data to be written
      END_STRUCT;
      ReadSDO : Struct   // management of a SDO read command
         fREQ : Bool := FALSE;   // flag controls REQ input of ReadSDO FB
         HW_ID : Hw_Io;   // hardware identifier of the accessed CM module in TIA Portal
         bSLOT : Byte;   // selected SLOT number
         iNODE : Int;   // CANopen node id of the accessed device
         wINDEX : Word;   // accessed index of the object dictionary
         bSUB : Byte;   // accessed subindex of the object dictionary
         diMaxSize : DInt;   // byte size of the destination area where to save the data
         fBusy : Bool;   // variable keeps the value of output BUSY of ReadSDO FB
         uiRet : UInt;   // variable keeps the value of output RET of ReadSDO FB
         uiSize : UInt;   // number of uploaded data bytes
         Data : "SDO_ReadData";   // data area where to copy the read data
      END_STRUCT;
   END_VAR
BEGIN
END_DATA_BLOCK

// folder: System blocks/Program resources

DATA_BLOCK "IEC_Timer_0_DB"   // DB2
{ S7_Optimized_Access := 'TRUE' }
AUTHOR : Simatic
FAMILY : IEC
NAME : IEC_TMR
VERSION : 1.0
// stored: InstanceOfName IEC_TIMER
"IEC_TIMER"
BEGIN
END_DATA_BLOCK

DATA_BLOCK "Timer_3.2"   // DB3
{ S7_Optimized_Access := 'TRUE' }
AUTHOR : Simatic
FAMILY : IEC
NAME : IEC_TMR
VERSION : 1.0
// stored: InstanceOfName IEC_TIMER
"IEC_TIMER"
BEGIN
END_DATA_BLOCK

// folder: (top level)

FUNCTION_BLOCK "Block_1"   // FB1, SCL
{ S7_Optimized_Access := 'TRUE' }
VERSION : 0.1
   VAR
      OptSen : Bool;
      MagSen : Bool;
      IndSen : Bool;
      CapSen : Bool;
      Delay : Time := T#1s;
      tank : Int;
      OccupyTimer : Bool;
      ReleaseT : Bool;
      NumPieces : Int;
      Man_Mode : Bool;
      Cyl_Down : Bool;
      Man_Move : Int;
      Errors : Word;
      temp : Int;
      Prev_State : UInt;
   END_VAR
BEGIN
   //IF "Swt1" = TRUE THEN //condition to enter manual mode
     //  IF "DB_State".State <> "MANUAL" THEN
          // "DB_State".State := "MANUAL";
      // END_IF;
   //END_IF;
   //

   #temp := ( BYTE_TO_INT("CANopenProcessImage".CM_PIInput.PIIn.TempHi) * 256) + BYTE_TO_INT("CANopenProcessImage".CM_PIInput.PIIn.TempLo);


   IF #temp > 27 THEN
       #Errors.%X7 := 1;
   END_IF;

   IF #Man_Mode = TRUE THEN //condition to enter manual mode
       IF "DB_State".State <> "MANUAL" THEN
           "DB_State".State := "MANUAL";
       END_IF;
   END_IF;

   IF "GlasLS" = FALSE THEN //Conditions to enter error state
       #Errors.%X1 := 1;
       "DB_State".State := "ERROR";
   END_IF;

   IF "EinLS" = TRUE THEN //Conditions to enter error state
       #Errors.%X2 := 1;
       "DB_State".State := "ERROR";
   END_IF;

   IF "Sonar_1" = TRUE OR "Sonar_2" = TRUE OR "Sonar_3" = TRUE  THEN //Conditions to enter error state
       #Errors.%X3 := 1;
       "DB_State".State := "ERROR";
   END_IF;

   IF "DB_State".State = "INIT" THEN
       #IndSen := FALSE;
       #CapSen := FALSE;
       #NumPieces := 0;
       #MagSen := FALSE; //Init vars
       #OptSen := FALSE;
       "ZylUp" := TRUE;
       "ZylDown" := FALSE;
       #Prev_State := 0;
       #tank := 0;
       #Errors := 0;

       IF "MagE_D" = FALSE THEN //Reset trolley
           "MCDIR" := 1;
           "MCGO" := 1;
           "Lampe_3" := "Clock_1Hz";
       ELSE //Begin test
           "MCDIR" := 0;
           "MCGO" := 0;
           "Lampe_3" := FALSE;
           "Lampe_2" := "Clock_1Hz";
           IF "Button_2" = 1 THEN
               "DB_State".State := "TEST";
           END_IF;
       END_IF;

   ELSIF "DB_State".State = "TEST" THEN
       "MCDIR" := 0;
       "MCGO" := 1;
       #Errors.%X5 := 1;
       "ZylDown" := FALSE;
       "ZendUP" := TRUE;
       "Lampe_3" := TRUE;
       "LED7" := TRUE;
       #Prev_State := "TEST";

       IF "Dist" < "tank1_dist" AND #tank < 1 THEN //Each of these are to check if our position s ok for the tank
           #Delay := T#1s;
           #tank := 1;
           "DB_State".State := "OCCUPIED";
       ELSIF "Dist" < "tank2_dist" AND #tank < 2 THEN
           #Delay := T#1s;
           #tank := 2;
           "DB_State".State := "OCCUPIED";
       ELSIF "Dist" < "tank3_dist" AND #tank < 3 THEN
           #Delay := T#1s;
           #tank := 3;
           "DB_State".State := "OCCUPIED";
       ELSIF "Dist" < "tank4_dist" AND #tank < 4 THEN
           #Delay := T#1s;
           #tank := 4;
           "DB_State".State := "OCCUPIED";
       ELSIF "MagE_U" = TRUE AND #tank < 5 THEN
               "DB_State".State := "RESET";
       END_IF;


   ELSIF "DB_State".State = "RESET" THEN
       "MCDIR" := 1;
       "MCGO" := 1;
       #tank := 0;
       "LED7" := FALSE;
       "LED6" := FALSE;
       "LED0" := FALSE;
       "LED1" := FALSE;
       "LED2" := FALSE;
       "LED3" := FALSE;
       "Lampe_3" := "Clock_1Hz";

       IF "MagE_D" = TRUE THEN //If we hit the end we reset the trolley and move on to the next state test/start
           "MCDIR" := 0;
           "MCGO" := 0;
           "Lampe_3" := FALSE;
           "Lampe_2" := "Clock_1Hz";
           IF "Button_2" = 1 THEN
               IF #Prev_State = "START" THEN
                   "DB_State".State := "TEST";
               ELSIF #Prev_State = "TEST" THEN
                   "DB_State".State := "START";
               END_IF;
           END_IF;
       END_IF;

   ELSIF "DB_State".State = "OCCUPIED" THEN
       "MCGO" := 0;
       "ZylDown" := TRUE;
       "ZylUp" := FALSE;


       IF #tank = 1 THEN //Set leds based on tank
           "LED0" := TRUE;
       ELSIF #tank = 2 THEN
           "LED1" := TRUE;
       ELSIF #tank = 3 THEN
           "LED2" := TRUE;
       ELSIF #tank = 4 THEN
           "LED3" := TRUE;
       END_IF;

       "IEC_Timer_0_DB".TON(IN := #OccupyTimer, //timer for cylinder
                            PT := #Delay,
                            Q => #ReleaseT);

       #OccupyTimer := TRUE;

       IF "IndNS_SS" = TRUE THEN // Get sensor data
           #IndSen := TRUE;
       END_IF;

       IF "KapNS" = TRUE THEN
           #CapSen := TRUE;
       END_IF;

       IF "ElMag" = TRUE THEN
           #MagSen := TRUE;
       END_IF;

       IF "OptNS" = TRUE THEN
           #OptSen := TRUE;
       END_IF;

       IF #ReleaseT = TRUE THEN
           "ZylDown" := FALSE;
           "ZylUp" := TRUE;
           "DB_State".State := #Prev_State;
           #ReleaseT := FALSE;
           #OccupyTimer := FALSE;
       END_IF;

   ELSIF "DB_State".State = "START" THEN
       "MCDIR" := 0;
       "MCGO" := 1;
       "ZylDown" := FALSE;
       #Errors.%X6 := 1;
       "ZendUP" := TRUE;
       "LED6" := TRUE;
       #Prev_State := "START"; 
       IF  #IndSen = TRUE  THEN //based on sensor data choose coating
           "DB_State".State := "COATING_A";
       ELSIF #OptSen = TRUE THEN
           "DB_State".State := "COATING_B";
       ELSE
           "DB_State".State := "COATING_C";
       END_IF;


   ELSIF "DB_State".State = "COATING_A" THEN //These states work similar to test
       IF "Dist" < "tank1_dist" AND #tank < 1 THEN
           #Delay := T#3s;
           #tank := 1;
           "DB_State".State := "OCCUPIED";
       ELSIF "Dist" < "tank4_dist" AND #tank < 2 THEN
           #Delay := T#3s;
           #tank := 4;
           "DB_State".State := "OCCUPIED";
       ELSIF "MagE_U" = TRUE AND #tank < 5 THEN
           #NumPieces := #NumPieces + 1;
           "DB_State".State := "RESET";
       END_IF;

   ELSIF "DB_State".State = "COATING_B" THEN
       IF "Dist" < "tank1_dist" AND #tank < 1 THEN
           #Delay := T#1s;
           #tank := 1;
           "DB_State".State := "OCCUPIED";
       ELSIF "Dist" < "tank3_dist" AND #tank < 2 THEN
           #tank := 3;
           #Delay := T#1s;
           "DB_State".State := "OCCUPIED";
       ELSIF "MagE_U" = TRUE AND #tank < 4 THEN
           #NumPieces := #NumPieces + 1;
           "DB_State".State := "RESET";
       END_IF;

   ELSIF "DB_State".State = "COATING_C" THEN
       IF "Dist" < "tank1_dist" AND #tank < 1 THEN
           #Delay := T#1s;
           #tank := 1;
           "DB_State".State := "OCCUPIED";
       ELSIF "Dist" < "tank2_dist" AND #tank < 2 THEN
           #Delay := T#2s;
           #tank := 2;
           "DB_State".State := "OCCUPIED";
       ELSIF "Dist" < "tank4_dist" AND #tank < 3 THEN
           #Delay := T#2s;
           #tank := 4;
           "DB_State".State := "OCCUPIED";
       ELSIF "MagE_U" = TRUE AND #tank < 5 THEN
           #NumPieces := #NumPieces + 1;
           "DB_State".State := "RESET";
       END_IF;

   ELSIF "DB_State".State = "MANUAL" THEN
       "Lampe_0" := "Clock_1Hz";
       "MCGO" := 0;
       "Lampe_3" := FALSE;

       //IF "Swt1" = FALSE THEN //get out of this state
           //"Lampe_0" := FALSE;
           //"DB_State".State := #Prev_State;
      // END_IF;

       IF #Man_Mode = FALSE THEN //get out of this state
           "Lampe_0" := FALSE;
           "DB_State".State := #Prev_State;
       END_IF;

       //IF "JOY_UpDown" > "Joy_Up" THEN //move trolley up/down
       IF #Man_Move = 1 THEN
           "Lampe_3" := TRUE;
           "MCGO" := 1;
           "MCDIR" := 0;
       //ELSIF "JOY_UpDown" < "Joy_Down" THEN
       ELSIF #Man_Move = -1 THEN
           "Lampe_3" := TRUE;
           "MCGO" := 1;
           "MCDIR" := 1;
       END_IF;

       //IF "Swt0" = TRUE THEN
       IF #Cyl_Down = TRUE THEN//push down cylinder based on location
           "Lampe_3" := TRUE;

           IF "Dist" < "tank1_dist" AND #tank < 1 THEN
               #tank := 1;
               "ZylDown" := TRUE;
               "ZylUp" := FALSE;
           ELSIF "Dist" < "tank2_dist" AND #tank < 2 THEN
               #tank := 2;
               "ZylDown" := TRUE;
               "ZylUp" := FALSE;
           ELSIF "Dist" < "tank3_dist" AND #tank < 3 THEN
               #tank := 3;
               "ZylDown" := TRUE;
               "ZylUp" := FALSE;
           ELSIF "Dist" < "tank4_dist" AND #tank < 4 THEN
               #tank := 4;
               "ZylDown" := TRUE;
               "ZylUp" := FALSE;
           ELSE
               #Errors.%X4 := 1;
               //"DB_State".State := "ERROR";
           END_IF;

       ELSE
           "Lampe_3" := FALSE;
           "ZylDown" := FALSE;
           "ZylUp" := TRUE;
       END_IF;

   ELSIF "DB_State".State = "ERROR" THEN
       "Lampe_0" := TRUE;
       "Lampe_3" := FALSE;
       "MCGO" := 0;
       IF "Button_0" = TRUE THEN
           "Lampe_0" := FALSE;
           #Errors := 0;
           IF #Prev_State = "START" THEN
               "DB_State".State := "START";// So after the reset it goes to test again
           ELSE
               //#Prev_State := "START";
               "DB_State".State := "RESET";
           END_IF;
       END_IF;

   END_IF;
END_FUNCTION_BLOCK

FUNCTION "Bsp3.1" : Void   // FC1, SCL
{ S7_Optimized_Access := 'TRUE' }
VERSION : 0.1
BEGIN
   IF "Swt0-7" <= 27 THEN
       "LED0-7" := "Swt0-7";
       ;
   ELSE
       "LED0-7" := 0;
   END_IF;
END_FUNCTION

FUNCTION "Bsp3.2" : Void   // FC2, SCL
{ S7_Optimized_Access := 'TRUE' }
VERSION : 0.1
BEGIN

   "Lampe_0" := "Clock_1Hz";
END_FUNCTION

FUNCTION "Bsp3.2_mit_timer" : Void   // FC3, SCL
{ S7_Optimized_Access := 'TRUE' }
VERSION : 0.1
BEGIN
   "Timer_3.2".TP(IN:="Clock_1Hz",
                  PT:=T#250ms,
                  Q=>"Lampe_0");
END_FUNCTION

FUNCTION "Bsp3.3" : Void   // FC4, SCL
{ S7_Optimized_Access := 'TRUE' }
VERSION : 0.1
   VAR CONSTANT
      JOY_MAX : Int := 1500;
      JOY_MIN : Int := -1500;
      JOY_MITTE : Int := 50;
   END_VAR
BEGIN
   IF "JOY_LeftRight" < 0.9 * #JOY_MIN THEN
       "LED3" := FALSE;
       "LED4" := FALSE;
       "LED5" := FALSE;
       "LED6" := TRUE;
   ELSIF "JOY_LeftRight" < 0.6 * #JOY_MIN THEN
       "LED3" := FALSE;
       "LED4" := FALSE;
       "LED5" := TRUE;
       "LED6" := FALSE;
   ELSIF "JOY_LeftRight" < 0.3 * #JOY_MIN THEN
       "LED3" := FALSE;
       "LED4" := TRUE;
       "LED5" := FALSE;
       "LED6" := FALSE;
   ELSIF "JOY_LeftRight" >= 0.3 * #JOY_MIN AND "JOY_LeftRight" <= #JOY_MITTE THEN
       "LED3" := TRUE;
       "LED4" := FALSE;
       "LED5" := FALSE;
       "LED6" := FALSE;
   ELSE
       "LED3" := FALSE;
       "LED4" := FALSE;
       "LED5" := FALSE;
       "LED6" := FALSE;
   END_IF;
END_FUNCTION

FUNCTION "Bsp3.4" : Void   // FC5, SCL
{ S7_Optimized_Access := 'TRUE' }
VERSION : 0.1
   VAR CONSTANT
      INT_MAX : Int := 16#FFFF;
   END_VAR
BEGIN
   //"MCSPEED" := #INT_MAX

   IF "DB_State".State = 0 THEN
       IF "MagE_D" = TRUE THEN
           "MCDIR" := 0;
           "DB_State".State := 1;
       ELSE
           "MCDIR" := 1;
           "DB_State".State := 2;
       END_IF;

   ELSIF "DB_State".State = 1 THEN
       "MCDIR" := 0;
       IF "MagE_U" = TRUE THEN
           "MCDIR" := 1;
           "DB_State".State := 2;

       END_IF;

   ELSIF "DB_State".State = 2 THEN
       "MCDIR" := 1;
       IF "MagE_D" = TRUE THEN
           "MCDIR" := 0;
           "DB_State".State := 1;

       END_IF;
   END_IF;

   IF "Swt7" THEN
       "MCGO" := TRUE;
       "Lampe_1" := FALSE;
       "Lampe_2" := TRUE;
      /// "DB_State".State := 0;
   ELSE
       "Lampe_1" := TRUE;
       "Lampe_2" := FALSE;
       "MCGO" := FALSE;
       //"DB_State".State := 10;
   END_IF;
END_FUNCTION

ORGANIZATION_BLOCK "Main"   // OB1, SCL, ProgramCycle
TITLE = "Main Program Sweep (Cycle)"
{ S7_Optimized_Access := 'TRUE' }
VERSION : 0.1
BEGIN

   "Block_1_DB"();
END_ORGANIZATION_BLOCK

ORGANIZATION_BLOCK "Startup"   // OB100, SCL, Startup
TITLE = "Complete Restart"
{ S7_Optimized_Access := 'TRUE' }
VERSION : 0.1
// initialization of all variables that are necessary for the demo
   VAR_INPUT
      LostRetentive : Bool;   // True if retentive data are lost
      LostRTC : Bool;   // True if date and time are lost
   END_VAR
BEGIN
   (* ------------------------------------------------------------------------
   Title:        initialize demo
   Description:  function initializes all variables to run the demo

   Author:       Christian Schlosser
   Version:      1.0
   Date:         2017-03-03
   ------------------------------------------------------------------------ *)

   ///////////////////////////////////////////////////////////////////////////
   // hardware identifier of the CM module in the PLC rack
   ///////////////////////////////////////////////////////////////////////////
   // see:
   //      Device Configuration
   //        / selected CM module
   //          / General
   //            / CANopen interface
   //              / Hardware identifier
   //
   // the hardware identifier is necessary for each communication with the
   // CM module:
   //    see chapter 8.1 CANopen interface functions:
   //        ID input of "Get Process Data In", "Set Process Data Out",
   //                    "SDO Read / Write", "Get Node & Network Status"
   //
   ///////////////////////////////////////////////////////////////////////////
   // note: hardware identifier of the CM module
   // -  TIA V13 provides the systen constant "Local~CM_CANopen_1"
   // -  TIA V14 does not provide this systen constant
   // => therefore "Local~CM_CANopen_1" is replaced by the actual value
   ///////////////////////////////////////////////////////////////////////////
   "Ctrl_CM_CANopen".HW_ID := 268; // "Local~CM_CANopen_1"; only valid for TIA V13

   ///////////////////////////////////////////////////////////////////////////
   // CANopen network
   ///////////////////////////////////////////////////////////////////////////
   // see: "Project Explorer" of the CM CANopen Configuration Studio
   //      of the demo project
   //
   // this demo uses constants to address 
   // - CM module
   //   node id of the CM module <=> "cNodeId_CM" 
   // - the single slaves
   //   - node id of the slave with node id 1 <=> "cNodeId_1"
   //   - node id of the slave with node id 2 <=> "cNodeId_2"
   //
   ///////////////////////////////////////////////////////////////////////////


   ///////////////////////////////////////////////////////////////////////////
   // "Get Process Data In"
   ///////////////////////////////////////////////////////////////////////////
   // - program group "Get Process Data In"
   //   provides all functionality to process the upload of the process image
   //   input from the CM module
   //   
   // - is realized by GetProcessDataIn [FC1]
   //   which is called in Network 2 of OB1
   //   
   // - the data are handled by
   //   - uploaded data from the CANopen network:
   //     => "CANopenProcessImage".CM_PIInput
   //        - data format: CANopen <=> little Endian
   //   - converted data to big endian:
   //     => "CANopenProcessImage".PLC_PIInput
   //        -  data format: PLC <=> big endian
   //     see UpdatePIInData_PLC[FC2]
   //     
   //   based on the structure "PIInput_CANopen"
   //   - "PIInput_CANopen"
   //     this structure reflects
   //           Configuration Studio / Process Image / Direction: IN
   //     it must also include the unused data bytes between data bytes
   //     that carry data !!!
   //
   // - the process image of the CM module is organized as a byte array
   //   the read process image input is a copy of this byte array from
   //   offset 0 up to offset i (i is discussed afterwards)
   //   -----------------------------------------------------------------
   //   | offset | Configuration Studio / Process Image / Direction: IN |
   //   ----------------------------------------------------------------- 
   //   |    0   |                    Address 0                         |
   //   ----------------------------------------------------------------- 
   //   |   ...  |                    Address ...                       |
   //   ----------------------------------------------------------------- 
   //   |    i   |                    Address i                         |
   //   ----------------------------------------------------------------- 
   //
   // - relationship between
   //   a) Configuration Studio / Process Image / Direction: IN
   //   b) bytes size of "PIInput_CANopen"
   //   c) TIA Portal / Device Configuration / CM module / General
   //        / CANopen interface / Module parameters: CANopen input data size
   //
   //   a) minimum byte size that covers all objects
   //      minimum byte size =   highest Address of Direction: IN
   //                          + byte size of the object at this Address
   //   b) "PIInput_CANopen" reflects Process Image / Direction: IN
   //      bytes size of "PIInput_CANopen" = minimum byte size
   //   c) CANopen input data size
   //      maximum number of data bytes that can be uploaded
   //      => CANopen input data size >= minimum byte size       
   //        
   //   note:
   //   any change of Process Image / Direction: IN requires that
   //   - the structure "PIInput_CANopen" must be adapted to Process Image / Direction: IN
   //   - "CANopenProcessImage".ByteSize_PIInput_CANopen
   //     - this variable keeps the byte size of the structure "PIInput_CANopen"
   //     - this variable must be adjusted 
   //   - CANopen input data size of the Module Parameter of the CM module in TIA Portal:
   //     must be checked if it still covers the minimum byte size
   //     
   // - "CANopenProcessImage".ByteSize_PIInput_CANopen
   //   - this variable keeps the byte size of "PIInput_CANopen"
   //   - this variable must be initialized
   //     because
   //       its value is passed to the input MLEN of RDREC
   //         which is called by GetProcessDataIn [FC1]
   //         - see "RDREC_GetProcessDataIn"()
   // 
   // - actual uploaded number of data bytes
   //   minimum of (value at the input MLEN) and (CANopen input data size)
   //
   ///////////////////////////////////////////////////////////////////////////
   // byte size of the structure "PIInput_CANopen"
   "CANopenProcessImage".ByteSize_PIInput_CANopen := 8; // demo: 20 bytes


   ///////////////////////////////////////////////////////////////////////////
   // "Set Process Data Out"
   ///////////////////////////////////////////////////////////////////////////
   // - program group "Set Process Data Out"
   //   provides all functionality to process the download of the process image
   //   output to the CM module
   //   
   // - is realized by SetProcessDataOut [FC3]
   //   which is called in Network 3 of OB1
   //
   // - the structure "Ctrl_CM_CANopen".SetPIOut
   //   controls the processing of "Set Process Data Out"
   //   
   // - the data are handled by
   //   - process image data of the PLC:
   //     => "CANopenProcessImage".PLC_PIOutput
   //        - data format: PLC <=> big Endian
   //   - converted and downloaded data to the CM module:
   //     => "CANopenProcessImage".CM_PIOutput
   //        -  data format: CANopen <=> little Endian
   //     see UpdatePIOutData_CM[FC4]
   //
   //   based on the structure "PIOutput_CANopen"
   //   - "PIOutput_CANopen"
   //     this structure reflects
   //           Configuration Studio / Process Image / Direction: OUT
   //     it must also include the unused data bytes between data bytes
   //     that carry data !!!
   //
   // - the process image of the CM module is organized as a byte array
   //   the downloaded process image output is copied as a byte array
   //   from offset 0 up to offset i (i is discussed afterwards)
   //   ------------------------------------------------------------------
   //   | offset | Configuration Studio / Process Image / Direction: OUT |
   //   ------------------------------------------------------------------ 
   //   |    0   |                    Address 0                          |
   //   ------------------------------------------------------------------ 
   //   |   ...  |                    Address ...                        |
   //   ------------------------------------------------------------------ 
   //   |    i   |                    Address i                          |
   //   ------------------------------------------------------------------ 
   //
   // - relationship between
   //   a) Configuration Studio / Process Image / Direction: OUT
   //   b) bytes size of "PIOutput_CANopen"
   //   c) TIA Portal / Device Configuration / CM module / General
   //        / CANopen interface / Module parameters: CANopen output data size
   //
   //   a) minimum byte size that covers all objects
   //      minimum byte size =   highest Address of Direction: OUT
   //                          + byte size of the object at this Address
   //   b) "PIOutput_CANopen" reflects Process Image / Direction: OUT
   //      => byte size of "PIOutput_CANopen" = minimum byte size
   //   c) CANopen output data size
   //      maximum number of data bytes that can be uploaded
   //      => CANopen output data size >= minimum byte size       
   //        
   //   note:
   //   any change of Process Image / Direction: OUT requires that
   //   - the structure "PIOutput_CANopen" must be adapted to Process Image / Direction: OUT
   //   - "CANopenProcessImage".ByteSize_PIOutput_CANopen
   //     - this variable keeps the byte size of the structure "PIOutput_CANopen"
   //     - this variable must be adjusted 
   //   - CANopen output data size of the Module Parameter of the CM module in TIA Portal:
   //     must be checked if it still covers the minimum byte size
   //     
   // - "CANopenProcessImage".ByteSize_PIOutput_CANopen
   //   - this variable keeps the byte size of "PIOutput_CANopen"
   //   - this variable must be initialized
   //     because
   //       its value is passed to the input LEN of WRREC
   //         which is called by SetProcessDataOut [FC3]
   //         - see "WRREC_SetProcessDataOut"()
   // 
   // - actual downloaded number of data bytes
   //   minimum of (value at the input LEN) and (CANopen output data size)
   //
   ///////////////////////////////////////////////////////////////////////////
   // byte size of the structure "PIOutput_CANopen"
   //"CANopenProcessImage".ByteSize_PIOutput_CANopen := 8; // demo: 16 bytes


   ///////////////////////////////////////////////////////////////////////////
   // "Get Node & Network Status"
   ///////////////////////////////////////////////////////////////////////////
   // - program group "Get Node & Network Status"
   //   provides all functionality to process "Get Node & Network Status"
   //   and to interpret the uploaded status informationen
   //   
   // - is realized by GetNodeNetworkStatus [FC18]
   //   which is called in Network 1 of OB1
   //
   // - the structure "Ctrl_CM_CANopen".GetNNStatus
   //   - controls the processing of "Get Node & Network Status"
   //   - provides the data area where the status information is saved
   //   
   ///////////////////////////////////////////////////////////////////////////


   ///////////////////////////////////////////////////////////////////////////
   // SDO Read
   ///////////////////////////////////////////////////////////////////////////
   // - program group "SDO Read"
   //   provides all functionality to process a SDO Read command
   //   and to interpret the read data 
   //   
   // - is realized by
   //   - SDORead_Request [FC6]
   //     which is called in Network 4 of OB1
   //     - checks if a SDO read command shall be processed
   //     - initializes the parameters of the SDO command
   //     - requests the processing of the SDO command
   //   - ReadSDO [FB104]
   //     which is called in Network 5 of OB1
   //     - processes the requested command
   //   - SDORead_InterpretReadData [FC7]
   //     which is called in Network 6 of OB1
   //     - analyses the result of the processed command
   //     - interprets the uploaded data
   //
   // - the structure "Ctrl_CM_CANopen".ReadSDO
   //   - controls the processing of "SDO Read"
   //   - holds the general information of the current SDO read command
   //   
   // - the read data are copied to the byte array
   //      "Ctrl_CM_CANopen".ReadSDO.Data
   //   according their order of reception
   //      "Ctrl_CM_CANopen".ReadSDO.Data.SDO_ReadData[1]: first data byte
   //      ...
   //      "Ctrl_CM_CANopen".ReadSDO.Data.SDO_ReadData[n]: n. data byte
   //
   ///////////////////////////////////////////////////////////////////////////


   ///////////////////////////////////////////////////////////////////////////
   // SDO Write
   ///////////////////////////////////////////////////////////////////////////
   // - program group "SDO Write"
   //   provides all functionality to process a SDO write command
   //   
   // - is realized by
   //   - SDOWrite_Request [FC5]
   //     which is called in Network 7 of OB1
   //     - checks if a SDO write command shall be processed
   //     - initializes the parameters of the SDO command
   //     - initializes the data that will be written
   //     - requests the processing of the SDO command
   //   - WriteSDO [FB105]
   //     which is called in Network 8 of OB1
   //     - processes the requested command
   //   - SDOWrite_InterpretResult [FC8]
   //     which is called in Network 9 of OB1
   //     - analyses the result of the processed command
   //
   // - the structure "Ctrl_CM_CANopen".WriteSDO
   //   - controls the processing of "SDO Write"
   //   - holds the general information of the current SDO Write command
   //   
   // - the data to be written are provided by the byte array
   //         "Ctrl_CM_CANopen".WriteSDO.Data.
   //   - "Ctrl_CM_CANopen".WriteSDO.Data.SDO_WriteData[1]: first transferred data byte
   //     ...
   //     "Ctrl_CM_CANopen".WriteSDO.Data.SDO_WriteData[n]: n. transferred data byte
   //
   ///////////////////////////////////////////////////////////////////////////


   ///////////////////////////////////////////////////////////////////////////
   // general hint: data
   ///////////////////////////////////////////////////////////////////////////
   // it must be differentiated between the data
   // - that are written to / read from the CM module
   // - that are used by the program to control the process
   // because
   // - the data exchange between the PLC and the CM module is done by
   //       WRREC / RDREC
   //   WRREC / RDREC request the transmission of an asynchronous telegram
   //   the transmission of the asynchronous telegram is not deterministic
   // to avoid
   // - that the written data are corrupted due to a change by the running program
   // - that the data that control the process are corrupted by the read data
   // 
   // demo:
   // - e.g.:
   //   - process image input data:
   //     - read data from the CM module :  "CANopenProcessImage".CM_PIInput
   //     - data to control the process  :  "CANopenProcessImage".PLC_PIInput
   //   - process image output data:
   //     - data to control the process  :  "CANopenProcessImage".PLC_PIOutput
   //     - written data to the CM module:  "CANopenProcessImage".CM_PIOutput
   //
   ///////////////////////////////////////////////////////////////////////////
END_ORGANIZATION_BLOCK

ORGANIZATION_BLOCK "Main_1"   // OB123, FBD, ProgramCycle
TITLE = "Main Program Sweep (Cycle)"
{ S7_Optimized_Access := 'TRUE' }
VERSION : 0.1
// demo application
BEGIN

REGION Network 1
   // demo: Get Node & Network Status
   // command is processed when InOutput REQ switches to TRUE and must stay TRUE
   // GetNodeNetworkStatus [FC18] automatically sets REQ to FALSE when the command has been processed
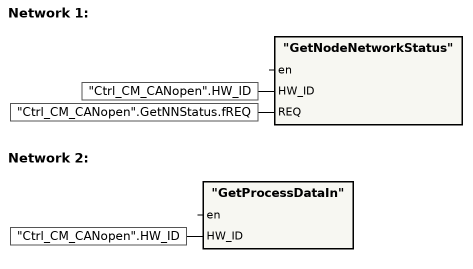
   "GetNodeNetworkStatus"(HW_ID := "Ctrl_CM_CANopen".HW_ID, REQ := "Ctrl_CM_CANopen".GetNNStatus.fREQ);
END_REGION

REGION Network 2
   // demo: Get Process Data In
   "GetProcessDataIn"(HW_ID := "Ctrl_CM_CANopen".HW_ID);
END_REGION

REGION Network 3
   // demo: Set Process Data Out
END_REGION

REGION Network 4
   // demo: check if a new SDO read command shall be processed:
   // if yes: initialize its parameters and request its execution
END_REGION

REGION Network 5
   // Process a SDO read command: 
   // note: a started a started SDO read command is processed until finish independent of REQ
   // REQ = TRUE: starts a SDO read command if ReadSDO FB is not occupied by a running SDO read command 
   // REQ = FALSE: - a started SDO read command is processed until finish independent of REQ
   //                          - no action if there is no running command
END_REGION

REGION Network 6
   // analyse the result and get the data of a processed SDO read command, ReadSDO FB shall not process a command
END_REGION

REGION Network 7
   // demo: run a requested SDO write command:
   // note: a started a started SDO write command is processed until finish independent of REQ
   // REQ = TRUE: starts a SDO write command if WriteSDO FB is not occupied by a running SDO write command 
   // REQ = FALSE: - a started SDO write command is processed until finish independent of REQ
   //                          - no action if there is no running command
END_REGION

REGION Network 8
   // analyse the result of the processed SDO write command, WriteSDO FB shall not process a command
END_REGION
END_ORGANIZATION_BLOCK

// folder: CM CANopen/Get Node & Network Status

FUNCTION "AnalyseNodeNetworkStatus" : Void   // FC14, SCL
{ S7_Optimized_Access := 'TRUE' }
VERSION : 0.1
   VAR_INPUT
      uiLen : UInt;   // number of uploaded bytes (condition: #fError = FALSE & #fVaild = TRUE)
   END_VAR
   VAR CONSTANT
      cOperatingMode : Byte := 16#0;   // Operating mode: CANopen Manager
   END_VAR
BEGIN
   (* ------------------------------------------------------------------------
   Title:        GetNNStatus_AnalyseResult
   Description:  function analyses the read "Get Node & Network Status"
                 function is exclusively called by GetNodeNetworkStatus [FC18]              

   Input:        uiLen   :  number of uploaded data bytes

   Output:       -

   Demo:         "Ctrl_CM_CANopen".GetNNStatus.abData provides all data
                 see input RECORD of "RDREC_GetNodeNetworkStatus"()

   Author:       Christian Schlosser
   Version:      1.0
   Date:         2017-03-03
   ------------------------------------------------------------------------ *)

   /////////////////////////////////////////////////////////////////////////
   // "Get Node & Network Status" has been processed sucessfully
   // - data are valid
   // - the first #uiLEN bytes of the byte array
   //      see input RECORD of "RDREC_GetNodeNetworkStatus"()
   //   contain data 
   /////////////////////////////////////////////////////////////////////////

   /////////////////////////////////////////////////////////////////////////
   //
   // discussion of the result:
   //
   /////////////////////////////////////////////////////////////////////////
   // valid data range
   /////////////////////////////////////////////////////////////////////////
   // "Ctrl_CM_CANopen".GetNNStatus.abData[0]
   // ...
   // "Ctrl_CM_CANopen".GetNNStatus.abData[#uiLen - 1]
   //
   /////////////////////////////////////////////////////////////////////////
   // Message error: "Ctrl_CM_CANopen".GetNNStatus.abData[0]
   /////////////////////////////////////////////////////////////////////////
   // "Ctrl_CM_CANopen".GetNNStatus.abData[0] <> 0
   // => error has reported by the CM module
   //    - see "Message Error Codes" on page 60 of the manual
   //    - ignore "Ctrl_CM_CANopen".GetNNStatus.abData[>0]
   //
   /////////////////////////////////////////////////////////////////////////
   // CANopen Module mode: "Ctrl_CM_CANopen".GetNNStatus.abData[3]
   /////////////////////////////////////////////////////////////////////////
   // Operating mode of the CM module
   //   0: CANopen Manager <=> Master
   //   1: CANopen slave   <=> Slave
   //   2: Transparent CAN
   //   
   // - this demo expects that the CM module is running in the CANopen
   //   Manager mode
   //   if the operating mode is not the expected one:
   //   => adjust:
   //      TIA Portal:
   //      Device configuration / Module parameters (of the CM module) / Operating mode
   //   => download the new hardware configuration to the PLC
   //   => Power Off / On the PLC
   //   
   //   hint:
   //   - demo expects that the CM module is running as CANopen Manager
   //     see constant #cOperatingMode
   //
   /////////////////////////////////////////////////////////////////////////
   // Error flags (module): "Ctrl_CM_CANopen".GetNNStatus.abData[1]
   /////////////////////////////////////////////////////////////////////////
   // - Bus off ( bit 0 ):
   //   possible reasons:
   //   - short cut of the CAN cable
   //   - the CAN network is not correctly terminated
   //     the CAN network must have a line topology  
   //   - wrong mounting of the CAN connection
   //   - the cable length is too long for the selected CAN baudrate
   //   - the CAN baudrate selected by the module parameters of the CM
   //     module is wrong
   //   - not every CANopen device in the CANopen network uses the selected
   //     CAN baudrate
   //
   //   note:
   //   - the CM module automatically retries to recover form bus off
   //
   //   action:
   //     -> check the above mentioned possible errors
   //
   //
   // - Configuration download error ( bit 1 ):
   //   the download of the CANopen configuration to the CM module
   //   has failed
   //   - the configuration of the CM module is invalid
   //
   //   action:
   //     -> download the CANopen configuration to the CM module
   //
   //
   // - Parameterization error ( bit 2 ):
   //   - the actual CANopen network does not match the configured / expected CANopen network
   //     possible reasons:
   //     - boot slave process of a slave has failed:
   //       possible error:
   //       - slave is missing
   //       - identity error
   //       - download of the configuration to the slave has failed
   //     - error control event of a slave:
   //       - timout of the heartbeat:
   //         slave has not transmitted its heartbeat within the configured heartbeat consumer time
   //       - timeout of the lifetime
   //         slave is guarded and has not responsed within its lifetime
   //       - heartbeat / guarding response of the slave reports another CANopen NMT state than expected
   //     - an unexpected device is present 
   //
   //    action:
   //    - analyse the status of each CANopen node id:
   //        "Ctrl_CM_CANopen".GetNNStatus.abData[5]   <=> status of CANopen node id 1
   //        ...
   //        "Ctrl_CM_CANopen".GetNNStatus.abData[131] <=> status of CANopen node id 127

   //
   // - NVS error ( bit 3 ):
   //   - the saved CANopen configuration is corrupted
   //   - the CM module does not communicate with the CANopen network
   //     RUN - CANopen LED: off
   //     ERR - CANopen LED: blinking with 1Hz
   //
   //   action:
   //     -> power off / on
   //     -> fatal error log can be read by SDO: index 5500h, subindex 1
   //        inform HMS
   //
   /////////////////////////////////////////////////////////////////////////
   // Error flags (network): "Ctrl_CM_CANopen".GetNNStatus.abData[2]
   /////////////////////////////////////////////////////////////////////////
   // - Network not ready ( bit 0 ):
   //   possible reasons:
   //   - CANopen Manager mode:
   //     - CM module is not operational:
   //       - network scan and initialization has not been finished
   //       - the CM module is disconnected from the CAN bus
   //       - error event of a slave
   //         - boot process of a slave has failed
   //         - slave is missing
   //         - error control event of a slave 
   //       - the CANopen state of the CM module has been changed
   //         by command
   //       - PLC is stopped
   //     - no slave is operational
   //
   //     action:
   //       -> check "CANopen Node status" <=> CANopen NMT status of the CM module
   //            "Ctrl_CM_CANopen".GetNNStatus.abData[4]
   //       -> check bit 1: node error control event
   //       -> analyse the status of each CANopen node id:
   //            "Ctrl_CM_CANopen".GetNNStatus.abData[5]   <=> status of CANopen node id 1
   //            ...
   //            "Ctrl_CM_CANopen".GetNNStatus.abData[131] <=> status of CANopen node id 127
   //
   //       additionally for more information:
   //       - read diagnostic object 5000h, subindex 2: CM CANopen state
   //       - read diagnostic object 5000h, subindex 1: Event indication
   //       see also chapter 7.3 Manufacturer Specific Objects
   //           in the manual of the CM Module
   //           all objects with 5xxxh index provide diagnostic information 
   //
   //   - CANopen slave mode:
   //     - CM module is not operational:
   //       - the CANopen state of the CM module has not been set to
   //         operational by the CANopen master
   //       - the CANopen state of the CM module has been changed by
   //         the CANopen master
   //       - the reaction to the following events is controlled by the
   //         configuration of the error behavior object:
   //         index 1029h, subindex 1:
   //              -> value = 0: enter pre-operational if operational
   //              -> value = 1: no change of NMT state
   //              -> value = 2: enter stopped
   //         events:
   //         - bus off
   //         - life guarding event (timeout of the guarding)
   //         - heartbeat event (timeout of consuming heartbeat)
   //         - received RPDO with less data than expected
   //         - received CAN message is lost (receive queue overrun)
   //         - transmit CAN message is lost (transmit queue overrun)
   //
   //       - the reaction to the following events is controlled by the
   //         configuration of the error behavior object:
   //         index 1029h, subindex 2:
   //              -> value = 0: enter pre-operational if operational
   //              -> value = 1: no change of NMT state
   //              -> value = 2: enter stopped
   //         events:
   //         - PLC is stopped
   //
   //     action:
   //        -> check "CANopen Node status"
   //             "Ctrl_CM_CANopen".GetNNStatus.abData[4]
   //        additionally for more information:
   //        - read diagnostic object 5000h, subindex 2: CM CANopen state
   //        - read diagnostic object 5000h, subindex 1: Event indication
   //        see also chapter 7.3 Manufacturer Specific Objects of the amanual
   //        - the objects 5003h - 5006h provide more diagnostic information:
   //          note:
   //          - another device only appears in one of these bitlists
   //            - if it has been entered in the consumer heartbeat list of the CM module
   //              and the configured consumer heartbeat time is not 0 
   //
   //
   // - Node error control event ( bit 1 ):
   //   possible reasons:
   //   - CANopen Manager mode:
   //     - error control event of a slave device
   //     - a slave is missing
   //     - identity error of a slave
   //     - download of the configuration of a slave has failed
   //       - the slave`s configuration generated by the CANopen Configuration Studio
   //         contains entries that are not supported by the slave
   //         or the data are not accepted by the slave  
   //         reason:
   //         - the EDS of the slave does not describe the real device
   //         - the device is not fully compliant to CANopen
   //     - a slave uses the node id of the CM module
   //     - present unexpected device:
   //       device is not entered in the Project Explorer of the CANopen Configuration
   //       Studio  
   //
   //     action:
   //       -> analyse the status of each CANopen node id:
   //            "Ctrl_CM_CANopen".GetNNStatus.abData[5]   <=> status of CANopen node id 1
   //            ...
   //            "Ctrl_CM_CANopen".GetNNStatus.abData[131] <=> status of CANopen node id 127
   //
   //   - CANopen slave mode:
   //     - timeout of the reception of the heartbeat of another CANopen
   //       device that is to be monitored:
   //         see index 1016h described in chapter 7.2 of the manual
   //
   //     action:
   //       -> read the diagnostic entry 5003h, subindex 1 - 4 of the
   //          CM module
   //            set bit marks the node id whose heartbeat is missing:
   //              subindex 1: bit i <=> node id: i +  1;  0 <= i <= 31
   //              subindex 2: bit i <=> node id: i + 33;  0 <= i <= 31
   //              subindex 3: bit i <=> node id: i + 65;  0 <= i <= 31
   //              subindex 2: bit i <=> node id: i + 97;  0 <= i <= 31
   //       -> read the diagnostic entry 5000h, subindex 1: Event indication
   //          set bit 13:
   //              check if the CM module is connected to the CAN bus
   //
   // - guarding error ( bit 2 ): only slave mode
   //   possible reasons:
   //   - guarding timeout:
   //     the master had started to guard the CM module but the next
   //     guarding request has not been received within
   //        life time factor (index 16#100D, subindex 0)
   //        * guard time     (index 16#100C, subindex 0)
   //
   /////////////////////////////////////////////////////////////////////////
   // CANopen Node Status: "Ctrl_CM_CANopen".GetNNStatus.abData[4]
   /////////////////////////////////////////////////////////////////////////
   //   CANopen status of the CM module:
   //   - NMT State Operational:
   //     CM module is operational
   //   - NMT State Unknown:
   //     CM module has not started its CANopen initialization after power on
   //     action:
   //       -> repeat "Get Node & Network Status"
   //   - Reset Node / Reset Communiation:
   //     CM module is processing its CANopen initialization
   //     action:
   //       -> repeat "Get Node & Network Status"
   //   - NMT State Stopped / NMT Pre-operational:
   //     CANopen Manager mode:
   //     - see above: Error flags (network): Network not ready
   //     CANopen slave mode:
   //     - see above: Error flags (network): Network not ready
   //
   /////////////////////////////////////////////////////////////////////////
   // "Network status":
   //          see manual: Offset     : 5
   //                      Data type  : Array of Uint8 (up to 127 elements)
   //                      Description: Network status
   // "Ctrl_CM_CANopen".GetNNStatus.abData[4 + node id]: 1 <= node id <= 127
   /////////////////////////////////////////////////////////////////////////
   //   - only CANopen Manager mode
   //     bits 0-3:
   //     - CANopen Device missing:
   //       - possible reasons:
   //         missing, error control event
   //         action:
   //           check if device is present
   //     - NMT State Operational:
   //       conditions:
   //       - device is operational
   //       - device must be controlled by the CM module:
   //              either by consuming heartbeat or by guarding
   //     - NMT State Unknown:
   //       if a device is not controlled by the CM module
   //              neither by consuming heartbeat nor by guarding
   //       its state is unknown:
   //              the error bits must be checked
   //
   //     bit 4: Configuration Error
   //     - possible reasons:
   //       - identity error
   //         the device is not the expected one:
   //         - the slave has reported another
   //             Device Type or Vendor-Id or Product Code or Revision Number
   //             or Serial Number
   //           than the expected one
   //         - an identity object is only checked if its value in the Configuration
   //           Studio is not 0:
   //           - see
   //             Network Management Configuration / Slave Assignment / Device Type
   //             Network Management Configuration / Slave Assignment / Vendor-ID
   //             Network Management Configuration / Slave Assignment / Product Code
   //             Network Management Configuration / Slave Assignment / Revision Number
   //             Network Management Configuration / Slave Assignment / Serial Number
   //
   //         note:
   //         - Device Type, Vendor-Id, Product Code and Serial Number must
   //           match exactly if checked
   //         - Revision Number:
   //           - major Revision Number (bits 16 - 31) must match
   //             exactly
   //           - the minor revision number (bits 0 - 15) must be greater
   //             or equal to the expected one in 1F87h, subindex slave`s CANopen node id
   //
   //       - concise DCF error
   //         see CM module object: 1F22h, subindex node id
   //         - the configuration of the slave does not match the object
   //           dictionary of the slave:
   //           the concise DCF contains an entry that causes an abort message
   //           of the booted slave:
   //           it must be checked
   //           - if the EDS of the slave really describes the device
   //           - if the slave is not implemented according CAnopen
   //         - the configuration is inconsistent( format error)
   //           should not happen
   //
   //       action: identity error and concise DCF error
   //         - read (SDO Read) the diagnostic entry "Event indication"
   //           index 5000h, subindex 1
   //           - the "Event indication" informs about the type of error:
   //             identity error:
   //               - indicated by MNCE (bit 3) and/or OIE (bit 4)
   //                 - action:
   //                     read (SDO Read) the diagnostic entry "Identity error
   //                     bit list": index 500Ah, subindex 1 - 4
   //             concise DCF error:
   //               - indicated by CONFIG_ERR (bit 10)
   //                 - action:
   //                     - read (SDO Read) the diagnostic entry "Wrong concise
   //                       DCF bit list": index 5009h, subindex 1 - 4
   //                     - log the CAN bus traffic and inform HMS
   //
   //                     - if "Wrong concise DCF bit list" does not report any
   //                       error:
   //                       read (SDO Read) the diagnostic entry "Inconsistent
   //                       concise DCF bit list": index 500Ah, subindex 1 - 4
   //                       inform HMS if the CANopen configuration has been
   //                       generated by the Configuration Studio
   //
   //             note index 5008h, 5009h and 500Ah:
   //               subindex 1: bit i <=> node id: i +  1;  0 <= i <= 31
   //               subindex 2: bit i <=> node id: i + 33;  0 <= i <= 31
   //               subindex 3: bit i <=> node id: i + 65;  0 <= i <= 31
   //               subindex 2: bit i <=> node id: i + 97;  0 <= i <= 31
   //
   //               set bit: error of the corresponding node id
   //
   //     bit 5: optional or mandatory slave
   //
   //     bit 7: present unexpected device
   //            1: this device is present but not expected in the CANopen network
   //
   /////////////////////////////////////////////////////////////////////////
   //
   // end of "discussion of the result"
   //
   /////////////////////////////////////////////////////////////////////////

   // function must be coded by the customer

   // check if "Message error" has occured
   IF "Ctrl_CM_CANopen".GetNNStatus.abData[0] <> 16#00 THEN
       // message error
       // see chapter 8.1.4 Get Node & Network Status
       //             Contents of Parameter RECORD: Offset 0
       // analysis of the message error code and reaction must be coded
       // by the customer
       ;

   // check operating mode of the CM module 
   ELSIF "Ctrl_CM_CANopen".GetNNStatus.abData[3] <> #cOperatingMode THEN
       // this is not the expected Operating mode
       // demo:
       //       expected: CANopen Manager mode
       ;

   // check if Error flags (module) reports an error
   // - bit 4 - 7: reserved
   ELSE // ELSIF "Ctrl_CM_CANopen".GetNNStatus.abData[3] <> #cOperatingMode THEN
       IF ("Ctrl_CM_CANopen".GetNNStatus.abData[1] & 16#0F) <> 16#00 THEN
           // bit 0: bus off
           // bit 1: configuration download error
           // bit 2: parameterization error
           // bit 3: NVS error in module
           ;
       END_IF;

       // check if Error flags (network) reports an error
       // - bit 3 - 7: reserved
       IF ("Ctrl_CM_CANopen".GetNNStatus.abData[2] & 16#07) <> 16#00 THEN
           // bit 0: network not ready
           // bit 1: node error control event
           // bit 2: guarding timeout of the master (only slave mode)
           ;
       END_IF;

       // check CANopen node status of the CM module: operational ?
       IF ("Ctrl_CM_CANopen".GetNNStatus.abData[4] <> 16#05) THEN
           // CM module is not operational
           ;
       END_IF;  

       // check Network status: 
       // - "Ctrl_CM_CANopen".GetNNStatus.abData[5]
       //   ...
       //   "Ctrl_CM_CANopen".GetNNStatus.abData[131]
       // - status of a single slave with CANopen node id x
       //   "Ctrl_CM_CANopen".GetNNStatus.abData[4 + x]
       //   
       //   note:
       //   - set Bit 4: analyse error
       //   - set Bit 7: unexpected device is present in the network
       //   - values of bits 0 - 3:
       //     - 0:    unknown
       //             hint:
       //                the CANopen NMT status of slave devices
       //                that are not controlled
       //                    - neither by consuming its heartbeat
       //                    - nor by active guarding
       //                cannot be displayed
       //                    - only its heartbeat or guarding reponse
       //                      informs about the CANopen NMT state
       //     - 1:     device is missing
       //     - 4,5,F: CANopen NMT status of the slave:
       //              its CANopen state can be displayed
       //              because the device is controlled by the CM module
       //                    - either by consuming its heartbeat
       //                    - or by active guarding
       //
       /////////////////////////////////////////////////////////////////////////

       ; // todo by the customer

   END_IF; // IF ... ELSIF ... ELSE
END_FUNCTION

FUNCTION "GetNodeNetworkStatus" : Void   // FC18, SCL
{ S7_Optimized_Access := 'TRUE' }
VERSION : 0.1
   VAR_INPUT
      HW_ID : Hw_Io;   // hardware identifier of the accessed CM module
   END_VAR
   VAR_IN_OUT
      REQ : Bool;   // TRUE: process Get Node & Network Status
   END_VAR
   VAR_TEMP
      fValid : Bool;
      fBusy : Bool;
      fError : Bool;
      dwStatus : DWord;
      uiLen : UInt;
   END_VAR
   VAR CONSTANT
      cByteSizeRecord : UInt := 131;   // byte size of "Ctrl_CM_CANopen".GetNNStatus.abData
   END_VAR
BEGIN
   (* ------------------------------------------------------------------------
   Title:        GetNodeNetworkStatus
   Description:  function
                 - checks if "Get Node & Network Status" has been requested
                 - processes the requested "Get Node & Network Status"
                 - calls AnalyseNodeNetworkStatus [FC14]
                   when the command has been processed and the data are valid                

   Input:        HW_ID:    hardware identifier of the accessed CM module
                           see:
                                Device Configuration
                                  / selected CM module
                                    / General
                                      / Hardware identifier

   InOut:        REQ:      TRUE:  run "Get Node & Network Status"
                                  - is automatically reset when the request
                                    has been processed
                           FALSE: do not run "Get Node & Network Status"

   Output:       -

   Demo:         "Ctrl_CM_CANopen".GetNNStatus.abData provides all data
                 see input RECORD of "RDREC_DB_GetNodeNetworkStatus"()

   Author:       Christian Schlosser
   Version:      1.0
   Date:         2017-03-03
   ------------------------------------------------------------------------ *)

   ///////////////////////////////////////////////////////////////////////////
   // check if "Get Node & network Status" is requested
   ///////////////////////////////////////////////////////////////////////////
   IF #REQ = FALSE THEN
       // no action
       // Get Node & Network Status has not been requested 
       RETURN;
   END_IF;

   ///////////////////////////////////////////////////////////////////////////
   // upload the node & network status
   ///////////////////////////////////////////////////////////////////////////
   "RDREC_GetNodeNetworkStatus"(REQ:=TRUE,
                                ID:=#HW_ID,
                                INDEX:=16#99, // see chapter 8.1.4 Get Node & Network Status
                                MLEN:=#cByteSizeRecord, // byte size of "Ctrl_CM_CANopen".GetNNStatus.abData
                                VALID=>#fValid,
                                BUSY=>#fBusy,
                                ERROR=>#fError,
                                STATUS=>#dwStatus,
                                LEN=>#uiLen,
                                RECORD:="Ctrl_CM_CANopen".GetNNStatus.abData);


   // check if command has been processed
   IF #fBusy = TRUE THEN
       // command is still running
       RETURN;
   END_IF;

   ///////////////////////////////////////////////////////////////////////////
   // command has been processed
   // - check result
   ///////////////////////////////////////////////////////////////////////////
   IF #fError = FALSE THEN
       // RDREC has not detected an error
       IF #fValid = TRUE THEN
           // data are valid
           "AnalyseNodeNetworkStatus"(#uiLen);
       ELSE
           // data are not valid
           // no action
           ;
       END_IF;
   ELSE
       // RDREC has detected an error
       // => #dwStatus must be analysed
       //    see online help: RDREC  
       //  => must be done by the customer
       ; // todo by the customer
   END_IF;

   ///////////////////////////////////////////////////////////////////////////
   // indicate that
   // - the requested "Node & Network Status" has been processed
   // - a new "Node & Network Status" can be requested
   ///////////////////////////////////////////////////////////////////////////
   // #REQ := FALSE; todo
END_FUNCTION

// folder: CM CANopen/Get Process Data In

FUNCTION "GetProcessDataIn" : Void   // FC6, SCL
{ S7_Optimized_Access := 'TRUE' }
VERSION : 0.1
   VAR_INPUT
      HW_ID : Hw_Io;   // hardware identifier of the accessed CM module
   END_VAR
   VAR_TEMP
      fValid : Bool;
      fBusy : Bool;
      fError : Bool;
      dwStatus : DWord;
      uiLen : UInt;
   END_VAR
BEGIN
   (* ------------------------------------------------------------------------
   Title:        GetProcessDataIn
   Description:  function
                 - uploades the process image input from the CM module
                 - calls UpdatePIInData_PLC [FC2]
                   which updates the according variables used by the PLC

                 hint:
                 it is recommented to differentiate between
                   - the data that are uploaded from the CM module
                   - the data the PLC works with
                 a) to avoid that PLC data is corrupted by the asynchronous
                    processing of the read telegram 
                 b) due to the different data format
                    - data format of the CM data:  little endian
                    - data format of the PLC data: big endian              


   Input:        HW_ID:    hardware identifier of the accessed CM module
                           see:
                                Device Configuration
                                  / selected CM module
                                    / General
                                      / Hardware identifier

   Output:       -

   Demo:         the uploaded data are copied to
                      "CANopenProcessImage".CM_PIInput
                 by RDREC   
                 the uploaded data are used to update the process image data
                 of the PLC
                      "CANopenProcessImage".PLC_PIInput 


   Author:       Christian Schlosser
   Version:      1.0
   Date:         2017-03-03
   ------------------------------------------------------------------------ *)

   ///////////////////////////////////////////////////////////////////////////
   // upload the process image input
   // 
   // hint: MLEN input of RDREC
   // - the process image of the CM module is organized as a byte array
   // - the read process image input is a copy of this byte array from
   //   -----------------------------------------------------------------
   //   | offset | Configuration Studio / Process Image / Direction: IN |
   //   ----------------------------------------------------------------- 
   //   |    0   |                    Address 0                         |
   //   ----------------------------------------------------------------- 
   //   |   ...  |                    Address ...                       |
   //   ----------------------------------------------------------------- 
   //   |    i   |                    Address i                         |
   //   ----------------------------------------------------------------- 
   //
   //   with i: minimum of "CANopen input data size" and MLEN 
   //
   //   with "CANopen input data size":
   //   - see TIA Portal:
   //     Device Configuration / selected CM module / General / Module parameters
   //     
   //   note:
   //   - data bytes within this range that do not contain data are also uploaded
   //   
   //   additional condition for MLEN:
   //   - MLEN <= byte size of the area where to copy the uploaded data
   // 
   ///////////////////////////////////////////////////////////////////////////
   "RDREC_GetProcessDataIn"(REQ:=TRUE,
                            ID:=#HW_ID,
                            INDEX:=16#90, // see chapter 8.1.1 Get Process Data In
                            MLEN:="CANopenProcessImage".ByteSize_PIInput_CANopen,
                            VALID=>#fValid,
                            BUSY=>#fBusy,
                            ERROR=>#fError,
                            STATUS=>#dwStatus,
                            LEN=>#uiLen,
                            RECORD:="CANopenProcessImage".CM_PIInput);

   // check if command has been processed
   IF #fBusy = TRUE THEN
       // command is still running
       RETURN;
   END_IF;

   ////////////////////////////////////////////////////////
   // command has been processed
   // - check result
   ////////////////////////////////////////////////////////
   IF #fError = FALSE THEN
       // RDREC was successful
       IF #fValid = TRUE THEN
           // data are valid
           // update the PI input data of the PLC
           // 
           // hint:
           // - it is recommented to differentiate between
           //     - the data that are uploaded from the CM module
           //     - the data the PLC works with
           //   a) to avoid that data is corrupted by the asynchronous
           //      processing of the read telegram 
           //   b) due to the different data format
           //      - data format of the CM data:  little endian
           //      - data format of the PLC data: big endian
           "UpdatePIInData_PLC"(#uiLen);

       ELSE
           // data are not valid
           // no action
           ;
       END_IF;
   ELSE
       // RDREC has detected an error
       // => #dwStatus must be analysed
       //    see online help: RDREC  
       //  => must be done by the customer
       ; // todo by the customer
   END_IF;
END_FUNCTION

FUNCTION "UpdatePIInData_PLC" : Void   // FC7, SCL
{ S7_Optimized_Access := 'TRUE' }
VERSION : 0.1
   VAR_INPUT
      uiLen : UInt;
   END_VAR
   VAR_TEMP
      dwHelp : DWord;
   END_VAR
BEGIN
   (* ------------------------------------------------------------------------
   Title:        UpdatePIInData_PLC
   Description:  function
                 - is called by GetProcessDataIn [FC1] when the process image
                   input data have been read from the CM module
                 - updates the data which are used by the application

                 hint:
                 it is recommented to differentiate between
                   - the data the PLC works with
                   - the data that are read from the CM module
                 a) to avoid that the PLC data is corrupted by the
                    asynchronous processing of the read telegram 
                 b) due to the different data format
                    - data format of the CM data:  little endian
                    - data format of the PLC data: big endian                            


                 hint:
                       function must be coded by the customer

   Input:        uiLen: number of read / uploaded data bytes

   InOut:        -

   Output:       -


   Demo:         the uploaded data are copied to
                      "CANopenProcessImage".CM_PIInput
                 these uploaded data are used to update the data
                 that are used by the application
                      "CANopenProcessImage".PLC_PIInput   


   Author:       Christian Schlosser
   Version:      1.0
   Date:         2017-03-03
   ------------------------------------------------------------------------ *)

   ///////////////////////////////////////////////////////////////////////////
   // hint: conversion of the data due to the different data format
   ///////////////////////////////////////////////////////////////////////////
   // - 8 bit values (Byte USInt, SInt):
   //   - must not be converted
   // - 16 bit values (Word, Int, UInt):
   //   - must be converted from big endian to little endian
   //     possible conversion:
   //     - SWAP function
   //     - PLC value.%B0 := CM value.%B1
   //       PLC value.%B1 := CM value.%B0
   // - 32 bit values (DWord, DInt, UDInt):
   //   - must be converted from big endian to little endian
   //     possible conversion:
   //     - SWAP function
   //     - PLC value.%B0 := CM value.%B3
   //       PLC value.%B1 := CM value.%B2
   //       PLC value.%B2 := CM value.%B1
   //       PLC value.%B3 := CM value.%B0
   // - Real (32 bit):
   //   - must be converted from big endian to little endian
   //     hint:
   //           this conversion cannot be done by
   //           - SWAP function
   //             => the returned values are not reliable
   //           - PLC value.%Bx
   //             => not possible for Real values
   //           therefore:
   //           the Real value must be converted first to DWORD
   //           see the method below
   //          
   //     1. convert Real to DWORD
   //        #dwhelp = REAL_TO_DWORD(CM real value);
   //     2. swap DWord value
   //        possible conversion:
   //        - SWAP function
   //     3. convert DWord to Real
   //        PLC real value = DWORD_TO_REAL(#dwhelp);
   //
   ///////////////////////////////////////////////////////////////////////////

   ///////////////////////////////////////////////////////////////////////////
   // hint: input uiLen
   ///////////////////////////////////////////////////////////////////////////
   // - uiLen informs about the number of uploaded data bytes
   // - the process image of the CM module is organized as a byte array
   // - the read process image input is a copy of this byte array from
   //   ---------------------------------------------------------------------
   //   |   offset   | Configuration Studio / Process Image / Direction: IN |
   //   ---------------------------------------------------------------------
   //   |      0     |                    Address 0                         |
   //   ---------------------------------------------------------------------
   //   |     ...    |                    Address ...                       |
   //   ---------------------------------------------------------------------
   //   | #uiLen - 1 |                    Address i                         |
   //   ---------------------------------------------------------------------
   // - uiLen can be used to check if the uploaded process iamge covers all
   //   data bytes that contain data
   //
   ///////////////////////////////////////////////////////////////////////////

   ///////////////////////////////////////////////////////////////////////////
   // update the data of the application
   ///////////////////////////////////////////////////////////////////////////
   // 8 bit values must not be swapped
   "CANopenProcessImage".PLC_PIInput.PIIn.TempLo :=
   "CANopenProcessImage".CM_PIInput.PIIn.TempLo;

   "CANopenProcessImage".PLC_PIInput.PIIn.TempHi :=
   "CANopenProcessImage".CM_PIInput.PIIn.TempHi;
END_FUNCTION

// ===== PLC "Target_1"  CPU 1214C DC/DC/DC =====

VAR_GLOBAL   // PLC tag table "Standard-Variablentabelle"
   "Swt0" AT %I0.0 : Bool;
   "Swt1" AT %I0.1 : Bool;
   "Swt2" AT %I0.2 : Bool;
   "Swt3" AT %I0.3 : Bool;
   "Swt4" AT %I0.4 : Bool;
   "Swt5" AT %I0.5 : Bool;
   "Swt6" AT %I0.6 : Bool;
   "Swt7" AT %I0.7 : Bool;
   "Swt0-7" AT %IB0 : Byte;
   "JOY_LeftRight" AT %IW70 : Int;
   "JOY_UpDown" AT %IW68 : Int;
   "MagE_D" AT %I7.1 : Bool;
   "MagE_U" AT %I7.2 : Bool;
   "Tast_1" AT %I2.2 : Bool;
   "LED0" AT %Q0.0 : Bool;
   "LED1" AT %Q0.1 : Bool;
   "LED2" AT %Q0.2 : Bool;
   "LED3" AT %Q0.3 : Bool;
   "LED4" AT %Q0.4 : Bool;
   "LED5" AT %Q0.5 : Bool;
   "LED6" AT %Q0.6 : Bool;
   "LED7" AT %Q0.7 : Bool;
   "LED0-7" AT %QB0 : Byte;
   "Lampe_0" AT %Q2.0 : Bool;
   "MCGO" AT %Q5.2 : Bool;
   "MCDIR" AT %Q5.3 : Bool;
   "MCSPEED" AT %QW66 : Word;
   "Lampe_1" AT %Q2.1 : Bool;
   "Lampe_2" AT %Q2.2 : Bool;
   "Clock_2.5Hz" AT %M8000.2 : Bool;
   "Clock_2Hz" AT %M8000.3 : Bool;
   "Clock_1.25Hz" AT %M8000.4 : Bool;
   "Clock_1Hz" AT %M8000.5 : Bool;
   "Clock_0.625Hz" AT %M8000.6 : Bool;
   "Clock_0.5Hz" AT %M8000.7 : Bool;
   "System_Byte" AT %MB8001 : Byte;
   "FirstScan" AT %M8001.0 : Bool;
   "AlwaysTRUE" AT %M8001.2 : Bool;
   "AlwaysFALSE" AT %M8001.3 : Bool;
   "IndNS_SS" AT %E9.0 : Bool;
   "IndNS_SSV" AT %E9.1 : Bool;
   "IndNS_OS" AT %I9.2 : Bool;
   "Dist" AT %EW74 : Word;
   "Druck" AT %EW72 : Word;
   "KapNS" AT %E5.2 : Bool;
   "ElMag" AT %A1.1 : Bool;
   "OptNS" AT %E5.3 : Bool;
   "ZendUP" AT %E8.1 : Bool;
   "ZendDO" AT %E8.0 : Bool;
END_VAR

VAR_GLOBAL CONSTANT   // PLC tag table "Standard-Variablentabelle"
   "CHECK" : UInt := 0;
   "INIT" : UInt := 1;
   "START" : UInt := 2;
   "PROCESS" : UInt := 3;
   "RUN" : UInt := 4;
END_VAR

DATA_BLOCK "DB_State"   // DB1
{ S7_Optimized_Access := 'TRUE' }
VERSION : 0.1
   VAR
      TimerFlag : Bool;
      "Timer" : Time;
      State : UInt;
   END_VAR
BEGIN
END_DATA_BLOCK

DATA_BLOCK "Block_1_DB"   // DB4
{ S7_Optimized_Access := 'TRUE' }
VERSION : 0.1
// stored: InstanceOfName Block_1
"Block_1"
BEGIN
END_DATA_BLOCK

// folder: System blocks/Program resources

DATA_BLOCK "Timer_3.2"   // DB2
{ S7_Optimized_Access := 'TRUE' }
AUTHOR : Simatic
FAMILY : IEC
NAME : IEC_TMR
VERSION : 1.0
// stored: InstanceOfName IEC_TIMER
"IEC_TIMER"
BEGIN
END_DATA_BLOCK

DATA_BLOCK "Timer_Cylinder"   // DB3
{ S7_Optimized_Access := 'TRUE' }
AUTHOR : Simatic
FAMILY : IEC
NAME : IEC_TMR
VERSION : 1.0
// stored: InstanceOfName IEC_TIMER
"IEC_TIMER"
BEGIN
END_DATA_BLOCK

